1742:L P[1218]  R[157] mm/sec CNT100 Offset,PR[24:Rotate_Offset] ;
1743:L P[1219]  R[157] mm/sec CNT100 Offset,PR[24:Rotate_Offset] ;
1744:L P[1220]  R[157] mm/sec CNT100 Offset,PR[24:Rotate_Offset] ;
1745:L P[1221]  R[157] mm/sec CNT100 Offset,PR[24:Rotate_Offset] ;
1746:L P[1222]  R[157] mm/sec CNT100 Offset,PR[24:Rotate_Offset] ;
1747:L P[1223]  R[157] mm/sec CNT100 Offset,PR[24:Rotate_Offset] ;
1748: !Pass74 ;
1749: LBL[174:Pass74] ;
1750:L P[1224]  R[157] mm/sec FINE Offset,PR[78:Offst_apprch]  ;
1751: WAIT   0.20(sec) ;
1752:L P[1224]  R[157] mm/sec CNT100 TA    0.00sec,CALL RUN_LASER_START Offset,PR[25:Start_Offset] ;
1754:L P[1225]  R[157] mm/sec CNT100 Offset,PR[24:Rotate_Offset] ;
1755:L P[1226]  R[157] mm/sec CNT100 TA    0.00sec,CALL RUN_LASER_STOP Offset,PR[26:Stop_Offset] ;
1757:L P[1226]  R[157] mm/sec FINE Offset,PR[76:Offst_dprt] ;
1758:L P[1227]  R[157] mm/sec CNT100 Offset,PR[24:Rotate_Offset] ;
1759:L P[1228]  R[157] mm/sec CNT100 Offset,PR[24:Rotate_Offset] ;
1760:L P[1229]  R[157] mm/sec CNT100 Offset,PR[24:Rotate_Offset] ;
1761:L P[1230]  R[157] mm/sec CNT100 Offset,PR[24:Rotate_Offset] ;
1762:L P[1231]  R[157] mm/sec CNT100 Offset,PR[24:Rotate_Offset] ;
1763:L P[1232]  R[157] mm/sec CNT100 Offset,PR[24:Rotate_Offset] ;
1764: !Pass75 ;
1765: LBL[175:Pass75] ;
1766:L P[1233]  R[157] mm/sec FINE Offset,PR[78:Offst_apprch]  ;
1767: WAIT   0.20(sec) ;
1768:L P[1233]  R[157] mm/sec CNT100 TA    0.00sec,CALL RUN_LASER_START Offset,PR[25:Start_Offset] ;
1770:L P[1234]  R[157] mm/sec CNT100 Offset,PR[24:Rotate_Offset] ;
1771:L P[1235]  R[157] mm/sec CNT100 TA    0.00sec,CALL RUN_LASER_STOP Offset,PR[26:Stop_Offset] ;
1773:L P[1235]  R[157] mm/sec FINE Offset,PR[76:Offst_dprt] ;
1774:L P[1236]  R[157] mm/sec CNT100 Offset,PR[24:Rotate_Offset] ;
1775:L P[1237]  R[157] mm/sec CNT100 Offset,PR[24:Rotate_Offset] ;
1776:L P[1238]  R[157] mm/sec CNT100 Offset,PR[24:Rotate_Offset] ;
1777:L P[1239]  R[157] mm/sec CNT100 Offset,PR[24:Rotate_Offset] ;
1778:L P[1240]  R[157] mm/sec CNT100 Offset,PR[24:Rotate_Offset] ;
1779:L P[1241]  R[157] mm/sec CNT100 Offset,PR[24:Rotate_Offset] ;
1780: !Pass76 ;
1781: LBL[176:Pass76] ;
1782:L P[1242]  R[157] mm/sec FINE Offset,PR[78:Offst_apprch]  ;
1783: WAIT   0.20(sec) ;
1784:L P[1242]  R[157] mm/sec CNT100 TA    0.00sec,CALL RUN_LASER_START Offset,PR[25:Start_Offset] ;
1786:L P[1243]  R[157] mm/sec CNT100 Offset,PR[24:Rotate_Offset] ;
1787:L P[1244]  R[157] mm/sec CNT100 Offset,PR[24:Rotate_Offset] ;
1788:L P[1245]  R[157] mm/sec CNT100 Offset,PR[24:Rotate_Offset] ;
1789:L P[1246]  R[157] mm/sec CNT100 Offset,PR[24:Rotate_Offset] ;
1790:L P[1247]  R[157] mm/sec CNT100 TA    0.00sec,CALL RUN_LASER_STOP Offset,PR[26:Stop_Offset] ;
1792:L P[1247]  R[157] mm/sec FINE Offset,PR[76:Offst_dprt] ;
1793:L P[1248]  R[157] mm/sec CNT100 Offset,PR[24:Rotate_Offset] ;
1794:L P[1249]  R[157] mm/sec CNT100 Offset,PR[24:Rotate_Offset] ;
1795:L P[1250]  R[157] mm/sec CNT100 Offset,PR[24:Rotate_Offset] ;
1796:L P[1251]  R[157] mm/sec CNT100 Offset,PR[24:Rotate_Offset] ;
1797:L P[1252]  R[157] mm/sec CNT100 Offset,PR[24:Rotate_Offset] ;
1798:L P[1253]  R[157] mm/sec CNT100 Offset,PR[24:Rotate_Offset] ;
1799: !Pass77 ;
1800: LBL[177:Pass77] ;
1801:L P[1254]  R[157] mm/sec FINE Offset,PR[78:Offst_apprch]  ;
1802: WAIT   0.20(sec) ;
1803:L P[1254]  R[157] mm/sec CNT100 TA    0.00sec,CALL RUN_LASER_START Offset,PR[25:Start_Offset] ;
1805:L P[1255]  R[157] mm/sec CNT100 Offset,PR[24:Rotate_Offset] ;
1806:L P[1256]  R[157] mm/sec CNT100 TA    0.00sec,CALL RUN_LASER_STOP Offset,PR[26:Stop_Offset] ;
1808:L P[1256]  R[157] mm/sec FINE Offset,PR[76:Offst_dprt] ;
1809:L P[1257]  R[157] mm/sec CNT100 Offset,PR[24:Rotate_Offset] ;
1810:L P[1258]  R[157] mm/sec CNT100 Offset,PR[24:Rotate_Offset] ;
1811:L P[1259]  R[157] mm/sec CNT100 Offset,PR[24:Rotate_Offset] ;
1812:L P[1260]  R[157] mm/sec CNT100 Offset,PR[24:Rotate_Offset] ;
1813:L P[1261]  R[157] mm/sec CNT100 Offset,PR[24:Rotate_Offset] ;
1814:L P[1262]  R[157] mm/sec CNT100 Offset,PR[24:Rotate_Offset] ;
1815: !Pass78 ;
1816: LBL[178:Pass78] ;
1817:L P[1263]  R[157] mm/sec FINE Offset,PR[78:Offst_apprch]  ;
1818: WAIT   0.20(sec) ;
1819:L P[1263]  R[157] mm/sec CNT100 TA    0.00sec,CALL RUN_LASER_START Offset,PR[25:Start_Offset] ;
1821:L P[1264]  R[157] mm/sec CNT100 Offset,PR[24:Rotate_Offset] ;
1822:L P[1265]  R[157] mm/sec CNT100 TA    0.00sec,CALL RUN_LASER_STOP Offset,PR[26:Stop_Offset] ;
1824:L P[1265]  R[157] mm/sec FINE Offset,PR[76:Offst_dprt] ;
1825:L P[1266]  R[157] mm/sec CNT100 Offset,PR[24:Rotate_Offset] ;
1826:L P[1267]  R[157] mm/sec CNT100 Offset,PR[24:Rotate_Offset] ;
1827:L P[1268]  R[157] mm/sec CNT100 Offset,PR[24:Rotate_Offset] ;
1828:L P[1269]  R[157] mm/sec CNT100 Offset,PR[24:Rotate_Offset] ;
1829:L P[1270]  R[157] mm/sec CNT100 Offset,PR[24:Rotate_Offset] ;
1830:L P[1271]  R[157] mm/sec CNT100 Offset,PR[24:Rotate_Offset] ;
1831: !Pass79 ;
1832: LBL[179:Pass79] ;
1833:L P[1272]  R[157] mm/sec FINE Offset,PR[78:Offst_apprch]  ;
1834: WAIT   0.20(sec) ;
1835:L P[1272]  R[157] mm/sec CNT100 TA    0.00sec,CALL RUN_LASER_START Offset,PR[25:Start_Offset] ;
1837:L P[1273]  R[157] mm/sec CNT100 Offset,PR[24:Rotate_Offset] ;
1838:L P[1274]  R[157] mm/sec CNT100 TA    0.00sec,CALL RUN_LASER_STOP Offset,PR[26:Stop_Offset] ;
1840:L P[1274]  R[157] mm/sec FINE Offset,PR[76:Offst_dprt] ;
1841:L P[1275]  R[157] mm/sec CNT100 Offset,PR[24:Rotate_Offset] ;
1842:L P[1276]  R[157] mm/sec CNT100 Offset,PR[24:Rotate_Offset] ;
1843:L P[1277]  R[157] mm/sec CNT100 Offset,PR[24:Rotate_Offset] ;
1844:L P[1278]  R[157] mm/sec CNT100 Offset,PR[24:Rotate_Offset] ;
1845:L P[1279]  R[157] mm/sec CNT100 Offset,PR[24:Rotate_Offset] ;
1846:L P[1280]  R[157] mm/sec CNT100 Offset,PR[24:Rotate_Offset] ;
1847: !Pass80 ;
1848: LBL[180:Pass80] ;
1849:L P[1281]  R[157] mm/sec FINE Offset,PR[78:Offst_apprch]  ;
1850: WAIT   0.20(sec) ;
1851:L P[1281]  R[157] mm/sec CNT100 TA    0.00sec,CALL RUN_LASER_START Offset,PR[25:Start_Offset] ;
1853:L P[1282]  R[157] mm/sec CNT100 Offset,PR[24:Rotate_Offset] ;
1854:L P[1283]  R[157] mm/sec CNT100 TA    0.00sec,CALL RUN_LASER_STOP Offset,PR[26:Stop_Offset] ;
1856:L P[1283]  R[157] mm/sec FINE Offset,PR[76:Offst_dprt] ;
1857:L P[1284]  R[157] mm/sec CNT100 Offset,PR[24:Rotate_Offset] ;
1858:L P[1285]  R[157] mm/sec CNT100 Offset,PR[24:Rotate_Offset] ;
1859:L P[1286]  R[157] mm/sec CNT100 Offset,PR[24:Rotate_Offset] ;
1860:L P[1287]  R[157] mm/sec CNT100 Offset,PR[24:Rotate_Offset] ;
1861:L P[1288]  R[157] mm/sec CNT100 Offset,PR[24:Rotate_Offset] ;
1862:L P[1289]  R[157] mm/sec CNT100 Offset,PR[24:Rotate_Offset] ;
1863: !Pass81 ;
1864: LBL[181:Pass81] ;
1865:L P[1290]  R[157] mm/sec FINE Offset,PR[78:Offst_apprch]  ;
1866: WAIT   0.20(sec) ;
1867:L P[1290]  R[157] mm/sec CNT100 TA    0.00sec,CALL RUN_LASER_START Offset,PR[25:Start_Offset] ;
1869:L P[1291]  R[157] mm/sec CNT100 Offset,PR[24:Rotate_Offset] ;
1870:L P[1292]  R[157] mm/sec CNT100 TA    0.00sec,CALL RUN_LASER_STOP Offset,PR[26:Stop_Offset] ;
1872:L P[1292]  R[157] mm/sec FINE Offset,PR[76:Offst_dprt] ;
1873:L P[1293]  R[157] mm/sec CNT100 Offset,PR[24:Rotate_Offset] ;
1874:L P[1294]  R[157] mm/sec CNT100 Offset,PR[24:Rotate_Offset] ;
1875:L P[1295]  R[157] mm/sec CNT100 Offset,PR[24:Rotate_Offset] ;
1876:L P[1296]  R[157] mm/sec CNT100 Offset,PR[24:Rotate_Offset] ;
1877:L P[1297]  R[157] mm/sec CNT100 Offset,PR[24:Rotate_Offset] ;
1878:L P[1298]  R[157] mm/sec CNT100 Offset,PR[24:Rotate_Offset] ;
1879: !Pass82 ;
1880: LBL[182:Pass82] ;
1881:L P[1299]  R[157] mm/sec FINE Offset,PR[78:Offst_apprch]  ;
1882: WAIT   0.20(sec) ;
1883:L P[1299]  R[157] mm/sec CNT100 TA    0.00sec,CALL RUN_LASER_START Offset,PR[25:Start_Offset] ;
1885:L P[1300]  R[157] mm/sec CNT100 Offset,PR[24:Rotate_Offset] ;
1886:L P[1301]  R[157] mm/sec CNT100 TA    0.00sec,CALL RUN_LASER_STOP Offset,PR[26:Stop_Offset] ;
1888:L P[1301]  R[157] mm/sec FINE Offset,PR[76:Offst_dprt] ;
1889:L P[1302]  R[157] mm/sec CNT100 Offset,PR[24:Rotate_Offset] ;
1890:L P[1303]  R[157] mm/sec CNT100 Offset,PR[24:Rotate_Offset] ;
1891:L P[1304]  R[157] mm/sec CNT100 Offset,PR[24:Rotate_Offset] ;
1892:L P[1305]  R[157] mm/sec CNT100 Offset,PR[24:Rotate_Offset] ;
1893:L P[1306]  R[157] mm/sec CNT100 Offset,PR[24:Rotate_Offset] ;
1894:L P[1307]  R[157] mm/sec CNT100 Offset,PR[24:Rotate_Offset] ;
1895: !Pass83 ;
1896: LBL[183:Pass83] ;
1897:L P[1308]  R[157] mm/sec FINE Offset,PR[78:Offst_apprch]  ;
1898: WAIT   0.20(sec) ;
1899:L P[1308]  R[157] mm/sec CNT100 TA    0.00sec,CALL RUN_LASER_START Offset,PR[25:Start_Offset] ;
1901:L P[1309]  R[157] mm/sec CNT100 Offset,PR[24:Rotate_Offset] ;
1902:L P[1310]  R[157] mm/sec CNT100 Offset,PR[24:Rotate_Offset] ;
1903:L P[1311]  R[157] mm/sec CNT100 Offset,PR[24:Rotate_Offset] ;
1904:L P[1312]  R[157] mm/sec CNT100 TA    0.00sec,CALL RUN_LASER_STOP Offset,PR[26:Stop_Offset] ;
1906:L P[1312]  R[157] mm/sec FINE Offset,PR[76:Offst_dprt] ;
1907:L P[1313]  R[157] mm/sec CNT100 Offset,PR[24:Rotate_Offset] ;
1908:L P[1314]  R[157] mm/sec CNT100 Offset,PR[24:Rotate_Offset] ;
1909:L P[1315]  R[157] mm/sec CNT100 Offset,PR[24:Rotate_Offset] ;
1910:L P[1316]  R[157] mm/sec CNT100 Offset,PR[24:Rotate_Offset] ;
1911:L P[1317]  R[157] mm/sec CNT100 Offset,PR[24:Rotate_Offset] ;
1912:L P[1318]  R[157] mm/sec CNT100 Offset,PR[24:Rotate_Offset] ;
1913: !Pass84 ;
1914: LBL[184:Pass84] ;
1915:L P[1319]  R[157] mm/sec FINE Offset,PR[78:Offst_apprch]  ;
1916: WAIT   0.20(sec) ;
1917:L P[1319]  R[157] mm/sec CNT100 TA    0.00sec,CALL RUN_LASER_START Offset,PR[25:Start_Offset] ;
1919:L P[1320]  R[157] mm/sec CNT100 Offset,PR[24:Rotate_Offset] ;
1920:L P[1321]  R[157] mm/sec CNT100 TA    0.00sec,CALL RUN_LASER_STOP Offset,PR[26:Stop_Offset] ;
1922:L P[1321]  R[157] mm/sec FINE Offset,PR[76:Offst_dprt] ;
1923:L P[1322]  R[157] mm/sec CNT100 Offset,PR[24:Rotate_Offset] ;
1924:L P[1323]  R[157] mm/sec CNT100 Offset,PR[24:Rotate_Offset] ;
1925:L P[1324]  R[157] mm/sec CNT100 Offset,PR[24:Rotate_Offset] ;
1926:L P[1325]  R[157] mm/sec CNT100 Offset,PR[24:Rotate_Offset] ;
1927:L P[1326]  R[157] mm/sec CNT100 Offset,PR[24:Rotate_Offset] ;
1928:L P[1327]  R[157] mm/sec CNT100 Offset,PR[24:Rotate_Offset] ;
1929: !Pass85 ;
1930: LBL[185:Pass85] ;
1931:L P[1328]  R[157] mm/sec FINE Offset,PR[78:Offst_apprch]  ;
1932: WAIT   0.20(sec) ;
1933:L P[1328]  R[157] mm/sec CNT100 TA    0.00sec,CALL RUN_LASER_START Offset,PR[25:Start_Offset] ;
1935:L P[1329]  R[157] mm/sec CNT100 Offset,PR[24:Rotate_Offset] ;
1936:L P[1330]  R[157] mm/sec CNT100 TA    0.00sec,CALL RUN_LASER_STOP Offset,PR[26:Stop_Offset] ;
1938:L P[1330]  R[157] mm/sec FINE Offset,PR[76:Offst_dprt] ;
1939:L P[1331]  R[157] mm/sec CNT100 Offset,PR[24:Rotate_Offset] ;
1940:L P[1332]  R[157] mm/sec CNT100 Offset,PR[24:Rotate_Offset] ;
1941:L P[1333]  R[157] mm/sec CNT100 Offset,PR[24:Rotate_Offset] ;
1942:L P[1334]  R[157] mm/sec CNT100 Offset,PR[24:Rotate_Offset] ;
1943:L P[1335]  R[157] mm/sec CNT100 Offset,PR[24:Rotate_Offset] ;
1944:L P[1336]  R[157] mm/sec CNT100 Offset,PR[24:Rotate_Offset] ;
1945: !Pass86 ;
1946: LBL[186:Pass86] ;
1947:L P[1337]  R[157] mm/sec FINE Offset,PR[78:Offst_apprch]  ;
1948: WAIT   0.20(sec) ;
1949:L P[1337]  R[157] mm/sec CNT100 TA    0.00sec,CALL RUN_LASER_START Offset,PR[25:Start_Offset] ;
1951:L P[1338]  R[157] mm/sec CNT100 Offset,PR[24:Rotate_Offset] ;
1952:L P[1339]  R[157] mm/sec CNT100 TA    0.00sec,CALL RUN_LASER_STOP Offset,PR[26:Stop_Offset] ;
1954:L P[1339]  R[157] mm/sec FINE Offset,PR[76:Offst_dprt] ;
1955:L P[1340]  R[157] mm/sec CNT100 Offset,PR[24:Rotate_Offset] ;
1956:L P[1341]  R[157] mm/sec CNT100 Offset,PR[24:Rotate_Offset] ;
1957:L P[1342]  R[157] mm/sec CNT100 Offset,PR[24:Rotate_Offset] ;
1958:L P[1343]  R[157] mm/sec CNT100 Offset,PR[24:Rotate_Offset] ;
1959:L P[1344]  R[157] mm/sec CNT100 Offset,PR[24:Rotate_Offset] ;
1960:L P[1345]  R[157] mm/sec CNT100 Offset,PR[24:Rotate_Offset] ;
1961: !Pass87 ;
1962: LBL[187:Pass87] ;
1963:L P[1346]  R[157] mm/sec FINE Offset,PR[78:Offst_apprch]  ;
1964: WAIT   0.20(sec) ;
1965:L P[1346]  R[157] mm/sec CNT100 TA    0.00sec,CALL RUN_LASER_START Offset,PR[25:Start_Offset] ;
1967:L P[1347]  R[157] mm/sec CNT100 Offset,PR[24:Rotate_Offset] ;
1968:L P[1348]  R[157] mm/sec CNT100 TA    0.00sec,CALL RUN_LASER_STOP Offset,PR[26:Stop_Offset] ;
1970:L P[1348]  R[157] mm/sec FINE Offset,PR[76:Offst_dprt] ;
1971:L P[1349]  R[157] mm/sec CNT100 Offset,PR[24:Rotate_Offset] ;
1972:L P[1350]  R[157] mm/sec CNT100 Offset,PR[24:Rotate_Offset] ;
1973:L P[1351]  R[157] mm/sec CNT100 Offset,PR[24:Rotate_Offset] ;
1974:L P[1352]  R[157] mm/sec CNT100 Offset,PR[24:Rotate_Offset] ;
1975:L P[1353]  R[157] mm/sec CNT100 Offset,PR[24:Rotate_Offset] ;
1976:L P[1354]  R[157] mm/sec CNT100 Offset,PR[24:Rotate_Offset] ;
1977: !Pass88 ;
1978: LBL[188:Pass88] ;
1979:L P[1355]  R[157] mm/sec FINE Offset,PR[78:Offst_apprch]  ;
1980: WAIT   0.20(sec) ;
1981:L P[1355]  R[157] mm/sec CNT100 TA    0.00sec,CALL RUN_LASER_START Offset,PR[25:Start_Offset] ;
1983:L P[1356]  R[157] mm/sec CNT100 Offset,PR[24:Rotate_Offset] ;
1984:L P[1357]  R[157] mm/sec CNT100 Offset,PR[24:Rotate_Offset] ;
1985:L P[1358]  R[157] mm/sec CNT100 Offset,PR[24:Rotate_Offset] ;
1986:L P[1359]  R[157] mm/sec CNT100 Offset,PR[24:Rotate_Offset] ;
1987:L P[1360]  R[157] mm/sec CNT100 TA    0.00sec,CALL RUN_LASER_STOP Offset,PR[26:Stop_Offset] ;
1989:L P[1360]  R[157] mm/sec FINE Offset,PR[76:Offst_dprt] ;
1990:L P[1361]  R[157] mm/sec CNT100 Offset,PR[24:Rotate_Offset] ;
1991:L P[1362]  R[157] mm/sec CNT100 Offset,PR[24:Rotate_Offset] ;
1992:L P[1363]  R[157] mm/sec CNT100 Offset,PR[24:Rotate_Offset] ;
1993:L P[1364]  R[157] mm/sec CNT100 Offset,PR[24:Rotate_Offset] ;
1994:L P[1365]  R[157] mm/sec CNT100 Offset,PR[24:Rotate_Offset] ;
1995:L P[1366]  R[157] mm/sec CNT100 Offset,PR[24:Rotate_Offset] ;
1996: !Pass89 ;
1997: LBL[189:Pass89] ;
1998:L P[1367]  R[157] mm/sec FINE Offset,PR[78:Offst_apprch]  ;
1999: WAIT   0.20(sec) ;
2000:L P[1367]  R[157] mm/sec CNT100 TA    0.00sec,CALL RUN_LASER_START Offset,PR[25:Start_Offset] ;
2002:L P[1368]  R[157] mm/sec CNT100 Offset,PR[24:Rotate_Offset] ;
2003:L P[1369]  R[157] mm/sec CNT100 Offset,PR[24:Rotate_Offset] ;
2004:L P[1370]  R[157] mm/sec CNT100 Offset,PR[24:Rotate_Offset] ;
2005:L P[1371]  R[157] mm/sec CNT100 TA    0.00sec,CALL RUN_LASER_STOP Offset,PR[26:Stop_Offset] ;
2007:L P[1371]  R[157] mm/sec FINE Offset,PR[76:Offst_dprt] ;
2008:L P[1372]  R[157] mm/sec CNT100 Offset,PR[24:Rotate_Offset] ;
2009:L P[1373]  R[157] mm/sec CNT100 Offset,PR[24:Rotate_Offset] ;
2010:L P[1374]  R[157] mm/sec CNT100 Offset,PR[24:Rotate_Offset] ;
2011:L P[1375]  R[157] mm/sec CNT100 Offset,PR[24:Rotate_Offset] ;
2012:L P[1376]  R[157] mm/sec CNT100 Offset,PR[24:Rotate_Offset] ;
2013:L P[1377]  R[157] mm/sec CNT100 Offset,PR[24:Rotate_Offset] ;
2014: !Pass90 ;
2015: LBL[190:Pass90] ;
2016:L P[1378]  R[157] mm/sec FINE Offset,PR[78:Offst_apprch]  ;
2017: WAIT   0.20(sec) ;
2018:L P[1378]  R[157] mm/sec CNT100 TA    0.00sec,CALL RUN_LASER_START Offset,PR[25:Start_Offset] ;
2020:L P[1379]  R[157] mm/sec CNT100 Offset,PR[24:Rotate_Offset] ;
2021:L P[1380]  R[157] mm/sec CNT100 Offset,PR[24:Rotate_Offset] ;
2022:L P[1381]  R[157] mm/sec CNT100 Offset,PR[24:Rotate_Offset] ;
2023:L P[1382]  R[157] mm/sec CNT100 TA    0.00sec,CALL RUN_LASER_STOP Offset,PR[26:Stop_Offset] ;
2025:L P[1382]  R[157] mm/sec FINE Offset,PR[76:Offst_dprt] ;
2026:L P[1383]  R[157] mm/sec CNT100 Offset,PR[24:Rotate_Offset] ;
2027:L P[1384]  R[157] mm/sec CNT100 Offset,PR[24:Rotate_Offset] ;
2028:L P[1385]  R[157] mm/sec CNT100 Offset,PR[24:Rotate_Offset] ;
2029:L P[1386]  R[157] mm/sec CNT100 Offset,PR[24:Rotate_Offset] ;
2030:L P[1387]  R[157] mm/sec CNT100 Offset,PR[24:Rotate_Offset] ;
2031:L P[1388]  R[157] mm/sec CNT100 Offset,PR[24:Rotate_Offset] ;
2032: !Pass91 ;
2033: LBL[191:Pass91] ;
2034:L P[1389]  R[157] mm/sec FINE Offset,PR[78:Offst_apprch]  ;
2035: WAIT   0.20(sec) ;
2036:L P[1389]  R[157] mm/sec CNT100 TA    0.00sec,CALL RUN_LASER_START Offset,PR[25:Start_Offset] ;
2038:L P[1390]  R[157] mm/sec CNT100 Offset,PR[24:Rotate_Offset] ;
2039:L P[1391]  R[157] mm/sec CNT100 TA    0.00sec,CALL RUN_LASER_STOP Offset,PR[26:Stop_Offset] ;
2041:L P[1391]  R[157] mm/sec FINE Offset,PR[76:Offst_dprt] ;
2042:L P[1392]  R[157] mm/sec CNT100 Offset,PR[24:Rotate_Offset] ;
2043:L P[1393]  R[157] mm/sec CNT100 Offset,PR[24:Rotate_Offset] ;
2044:L P[1394]  R[157] mm/sec CNT100 Offset,PR[24:Rotate_Offset] ;
2045:L P[1395]  R[157] mm/sec CNT100 Offset,PR[24:Rotate_Offset] ;
2046:L P[1396]  R[157] mm/sec CNT100 Offset,PR[24:Rotate_Offset] ;
2047:L P[1397]  R[157] mm/sec CNT100 Offset,PR[24:Rotate_Offset] ;
2048: !Pass92 ;
2049: LBL[192:Pass92] ;
2050:L P[1398]  R[157] mm/sec FINE Offset,PR[78:Offst_apprch]  ;
2051: WAIT   0.20(sec) ;
2052:L P[1398]  R[157] mm/sec CNT100 TA    0.00sec,CALL RUN_LASER_START Offset,PR[25:Start_Offset] ;
2054:L P[1399]  R[157] mm/sec CNT100 Offset,PR[24:Rotate_Offset] ;
2055:L P[1400]  R[157] mm/sec CNT100 TA    0.00sec,CALL RUN_LASER_STOP Offset,PR[26:Stop_Offset] ;
2057:L P[1400]  R[157] mm/sec FINE Offset,PR[76:Offst_dprt] ;
2058:L P[1401]  R[157] mm/sec CNT100 Offset,PR[24:Rotate_Offset] ;
2059:L P[1402]  R[157] mm/sec CNT100 Offset,PR[24:Rotate_Offset] ;
2060:L P[1403]  R[157] mm/sec CNT100 Offset,PR[24:Rotate_Offset] ;
2061:L P[1404]  R[157] mm/sec CNT100 Offset,PR[24:Rotate_Offset] ;
2062:L P[1405]  R[157] mm/sec CNT100 Offset,PR[24:Rotate_Offset] ;
2063:L P[1406]  R[157] mm/sec CNT100 Offset,PR[24:Rotate_Offset] ;
2064: !Pass93 ;
2065: LBL[193:Pass93] ;
2066:L P[1407]  R[157] mm/sec FINE Offset,PR[78:Offst_apprch]  ;
2067: WAIT   0.20(sec) ;
2068:L P[1407]  R[157] mm/sec CNT100 TA    0.00sec,CALL RUN_LASER_START Offset,PR[25:Start_Offset] ;
2070:L P[1408]  R[157] mm/sec CNT100 Offset,PR[24:Rotate_Offset] ;
2071:L P[1409]  R[157] mm/sec CNT100 Offset,PR[24:Rotate_Offset] ;
2072:L P[1410]  R[157] mm/sec CNT100 Offset,PR[24:Rotate_Offset] ;
2073:L P[1411]  R[157] mm/sec CNT100 Offset,PR[24:Rotate_Offset] ;
2074:L P[1412]  R[157] mm/sec CNT100 Offset,PR[24:Rotate_Offset] ;
2075:L P[1413]  R[157] mm/sec CNT100 Offset,PR[24:Rotate_Offset] ;
2076:L P[1414]  R[157] mm/sec CNT100 Offset,PR[24:Rotate_Offset] ;
2077:L P[1415]  R[157] mm/sec CNT100 Offset,PR[24:Rotate_Offset] ;
2078:L P[1416]  R[157] mm/sec CNT100 Offset,PR[24:Rotate_Offset] ;
2079:L P[1417]  R[157] mm/sec CNT100 TA    0.00sec,CALL RUN_LASER_STOP Offset,PR[26:Stop_Offset] ;
2081:L P[1417]  R[157] mm/sec FINE Offset,PR[76:Offst_dprt] ;
2082:L P[1418]  R[157] mm/sec CNT100 Offset,PR[24:Rotate_Offset] ;
2083:L P[1419]  R[157] mm/sec CNT100 Offset,PR[24:Rotate_Offset] ;
2084:L P[1420]  R[157] mm/sec CNT100 Offset,PR[24:Rotate_Offset] ;
2085:L P[1421]  R[157] mm/sec CNT100 Offset,PR[24:Rotate_Offset] ;
2086:L P[1422]  R[157] mm/sec CNT100 Offset,PR[24:Rotate_Offset] ;
2087:L P[1423]  R[157] mm/sec CNT100 Offset,PR[24:Rotate_Offset] ;
2088: !Pass94 ;
2089: LBL[194:Pass94] ;
2090:L P[1424]  R[157] mm/sec FINE Offset,PR[78:Offst_apprch]  ;
2091: WAIT   0.20(sec) ;
2092:L P[1424]  R[157] mm/sec CNT100 TA    0.00sec,CALL RUN_LASER_START Offset,PR[25:Start_Offset] ;
2094:L P[1425]  R[157] mm/sec CNT100 Offset,PR[24:Rotate_Offset] ;
2095:L P[1426]  R[157] mm/sec CNT100 Offset,PR[24:Rotate_Offset] ;
2096:L P[1427]  R[157] mm/sec CNT100 Offset,PR[24:Rotate_Offset] ;
2097:L P[1428]  R[157] mm/sec CNT100 Offset,PR[24:Rotate_Offset] ;
2098:L P[1429]  R[157] mm/sec CNT100 TA    0.00sec,CALL RUN_LASER_STOP Offset,PR[26:Stop_Offset] ;
2100:L P[1429]  R[157] mm/sec FINE Offset,PR[76:Offst_dprt] ;
2101:L P[1430]  R[157] mm/sec CNT100 Offset,PR[24:Rotate_Offset] ;
2102:L P[1431]  R[157] mm/sec CNT100 Offset,PR[24:Rotate_Offset] ;
2103:L P[1432]  R[157] mm/sec CNT100 Offset,PR[24:Rotate_Offset] ;
2104:L P[1433]  R[157] mm/sec CNT100 Offset,PR[24:Rotate_Offset] ;
2105:L P[1434]  R[157] mm/sec CNT100 Offset,PR[24:Rotate_Offset] ;
2106:L P[1435]  R[157] mm/sec CNT100 Offset,PR[24:Rotate_Offset] ;
2107: !Pass95 ;
2108: LBL[195:Pass95] ;
2109:L P[1436]  R[157] mm/sec FINE Offset,PR[78:Offst_apprch]  ;
2110: WAIT   0.20(sec) ;
2111:L P[1436]  R[157] mm/sec CNT100 TA    0.00sec,CALL RUN_LASER_START Offset,PR[25:Start_Offset] ;
2113:L P[1437]  R[157] mm/sec CNT100 Offset,PR[24:Rotate_Offset] ;
2114:L P[1438]  R[157] mm/sec CNT100 Offset,PR[24:Rotate_Offset] ;
2115:L P[1439]  R[157] mm/sec CNT100 Offset,PR[24:Rotate_Offset] ;
2116:L P[1440]  R[157] mm/sec CNT100 TA    0.00sec,CALL RUN_LASER_STOP Offset,PR[26:Stop_Offset] ;
2118:L P[1440]  R[157] mm/sec FINE Offset,PR[76:Offst_dprt] ;
2119:L P[1441]  R[157] mm/sec CNT100 Offset,PR[24:Rotate_Offset] ;
2120:L P[1442]  R[157] mm/sec CNT100 Offset,PR[24:Rotate_Offset] ;
2121:L P[1443]  R[157] mm/sec CNT100 Offset,PR[24:Rotate_Offset] ;
2122:L P[1444]  R[157] mm/sec CNT100 Offset,PR[24:Rotate_Offset] ;
2123:L P[1445]  R[157] mm/sec CNT100 Offset,PR[24:Rotate_Offset] ;
2124:L P[1446]  R[157] mm/sec CNT100 Offset,PR[24:Rotate_Offset] ;
2125: !Pass96 ;
2126: LBL[196:Pass96] ;
2127:L P[1447]  R[157] mm/sec FINE Offset,PR[78:Offst_apprch]  ;
2128: WAIT   0.20(sec) ;
2129:L P[1447]  R[157] mm/sec CNT100 TA    0.00sec,CALL RUN_LASER_START Offset,PR[25:Start_Offset] ;
2131:L P[1448]  R[157] mm/sec CNT100 Offset,PR[24:Rotate_Offset] ;
2132:L P[1449]  R[157] mm/sec CNT100 Offset,PR[24:Rotate_Offset] ;
2133:L P[1450]  R[157] mm/sec CNT100 Offset,PR[24:Rotate_Offset] ;
2134:L P[1451]  R[157] mm/sec CNT100 TA    0.00sec,CALL RUN_LASER_STOP Offset,PR[26:Stop_Offset] ;
2136:L P[1451]  R[157] mm/sec FINE Offset,PR[76:Offst_dprt] ;
2137:L P[1452]  R[157] mm/sec CNT100 Offset,PR[24:Rotate_Offset] ;
2138:L P[1453]  R[157] mm/sec CNT100 Offset,PR[24:Rotate_Offset] ;
2139:L P[1454]  R[157] mm/sec CNT100 Offset,PR[24:Rotate_Offset] ;
2140:L P[1455]  R[157] mm/sec CNT100 Offset,PR[24:Rotate_Offset] ;
2141:L P[1456]  R[157] mm/sec CNT100 Offset,PR[24:Rotate_Offset] ;
2142:L P[1457]  R[157] mm/sec CNT100 Offset,PR[24:Rotate_Offset] ;
2143: !Pass97 ;
2144: LBL[197:Pass97] ;
2145:L P[1458]  R[157] mm/sec FINE Offset,PR[78:Offst_apprch]  ;
2146: WAIT   0.20(sec) ;
2147:L P[1458]  R[157] mm/sec CNT100 TA    0.00sec,CALL RUN_LASER_START Offset,PR[25:Start_Offset] ;
2149:L P[1459]  R[157] mm/sec CNT100 Offset,PR[24:Rotate_Offset] ;
2150:L P[1460]  R[157] mm/sec CNT100 Offset,PR[24:Rotate_Offset] ;
2151:L P[1461]  R[157] mm/sec CNT100 Offset,PR[24:Rotate_Offset] ;
2152:L P[1462]  R[157] mm/sec CNT100 TA    0.00sec,CALL RUN_LASER_STOP Offset,PR[26:Stop_Offset] ;
2154:L P[1462]  R[157] mm/sec FINE Offset,PR[76:Offst_dprt] ;
2155:L P[1463]  R[157] mm/sec CNT100 Offset,PR[24:Rotate_Offset] ;
2156:L P[1464]  R[157] mm/sec CNT100 Offset,PR[24:Rotate_Offset] ;
2157:L P[1465]  R[157] mm/sec CNT100 Offset,PR[24:Rotate_Offset] ;
2158:L P[1466]  R[157] mm/sec CNT100 Offset,PR[24:Rotate_Offset] ;
2159:L P[1467]  R[157] mm/sec CNT100 Offset,PR[24:Rotate_Offset] ;
2160:L P[1468]  R[157] mm/sec CNT100 Offset,PR[24:Rotate_Offset] ;
2161: !Pass98 ;
2162: LBL[198:Pass98] ;
2163:L P[1469]  R[157] mm/sec FINE Offset,PR[78:Offst_apprch]  ;
2164: WAIT   0.20(sec) ;
2165:L P[1469]  R[157] mm/sec CNT100 TA    0.00sec,CALL RUN_LASER_START Offset,PR[25:Start_Offset] ;
2167:L P[1470]  R[157] mm/sec CNT100 Offset,PR[24:Rotate_Offset] ;
2168:L P[1471]  R[157] mm/sec CNT100 Offset,PR[24:Rotate_Offset] ;
2169:L P[1472]  R[157] mm/sec CNT100 Offset,PR[24:Rotate_Offset] ;
2170:L P[1473]  R[157] mm/sec CNT100 TA    0.00sec,CALL RUN_LASER_STOP Offset,PR[26:Stop_Offset] ;
2172:L P[1473]  R[157] mm/sec FINE Offset,PR[76:Offst_dprt] ;
2173:L P[1474]  R[157] mm/sec CNT100 Offset,PR[24:Rotate_Offset] ;
2174:L P[1475]  R[157] mm/sec CNT100 Offset,PR[24:Rotate_Offset] ;
2175:L P[1476]  R[157] mm/sec CNT100 Offset,PR[24:Rotate_Offset] ;
2176:L P[1477]  R[157] mm/sec CNT100 Offset,PR[24:Rotate_Offset] ;
2177:L P[1478]  R[157] mm/sec CNT100 Offset,PR[24:Rotate_Offset] ;
2178:L P[1479]  R[157] mm/sec CNT100 Offset,PR[24:Rotate_Offset] ;
2179: !Pass99 ;
2180: LBL[199:Pass99] ;
2181:L P[1480]  R[157] mm/sec FINE Offset,PR[78:Offst_apprch]  ;
2182: WAIT   0.20(sec) ;
2183:L P[1480]  R[157] mm/sec CNT100 TA    0.00sec,CALL RUN_LASER_START Offset,PR[25:Start_Offset] ;
2185:L P[1481]  R[157] mm/sec CNT100 Offset,PR[24:Rotate_Offset] ;
2186:L P[1482]  R[157] mm/sec CNT100 TA    0.00sec,CALL RUN_LASER_STOP Offset,PR[26:Stop_Offset] ;
2188:L P[1482]  R[157] mm/sec FINE Offset,PR[76:Offst_dprt] ;
2189:L P[1483]  R[157] mm/sec CNT100 Offset,PR[24:Rotate_Offset] ;
2190:L P[1484]  R[157] mm/sec CNT100 Offset,PR[24:Rotate_Offset] ;
2191:L P[1485]  R[157] mm/sec CNT100 Offset,PR[24:Rotate_Offset] ;
2192:L P[1486]  R[157] mm/sec CNT100 Offset,PR[24:Rotate_Offset] ;
2193:L P[1487]  R[157] mm/sec CNT100 Offset,PR[24:Rotate_Offset] ;
2194:L P[1488]  R[157] mm/sec CNT100 Offset,PR[24:Rotate_Offset] ;
2195: !Pass100 ;
2196: LBL[1100:Pass100] ;
2197:L P[1489]  R[157] mm/sec FINE Offset,PR[78:Offst_apprch]  ;
2198: WAIT   0.20(sec) ;
2199:L P[1489]  R[157] mm/sec CNT100 TA    0.00sec,CALL RUN_LASER_START Offset,PR[25:Start_Offset] ;
2201:L P[1490]  R[157] mm/sec CNT100 Offset,PR[24:Rotate_Offset] ;
2202:L P[1491]  R[157] mm/sec CNT100 TA    0.00sec,CALL RUN_LASER_STOP Offset,PR[26:Stop_Offset] ;
2204:L P[1491]  R[157] mm/sec FINE Offset,PR[76:Offst_dprt] ;
2205:L P[1492]  R[157] mm/sec CNT100 Offset,PR[24:Rotate_Offset] ;
2206:L P[1493]  R[157] mm/sec CNT100 Offset,PR[24:Rotate_Offset] ;
2207:L P[1494]  R[157] mm/sec CNT100 Offset,PR[24:Rotate_Offset] ;
2208:L P[1495]  R[157] mm/sec CNT100 Offset,PR[24:Rotate_Offset] ;
2209:L P[1496]  R[157] mm/sec CNT100 Offset,PR[24:Rotate_Offset] ;
2210:L P[1497]  R[157] mm/sec CNT100 Offset,PR[24:Rotate_Offset] ;
2211: !Pass101 ;
2212: LBL[1101:Pass101] ;
2213:L P[1498]  R[157] mm/sec FINE Offset,PR[78:Offst_apprch]  ;
2214: WAIT   0.20(sec) ;
2215:L P[1498]  R[157] mm/sec CNT100 TA    0.00sec,CALL RUN_LASER_START Offset,PR[25:Start_Offset] ;
2217:L P[1499]  R[157] mm/sec CNT100 Offset,PR[24:Rotate_Offset] ;
2218:L P[1500]  R[157] mm/sec CNT100 Offset,PR[24:Rotate_Offset] ;
2219:L P[1501]  R[157] mm/sec CNT100 Offset,PR[24:Rotate_Offset] ;
2220:L P[1502]  R[157] mm/sec CNT100 TA    0.00sec,CALL RUN_LASER_STOP Offset,PR[26:Stop_Offset] ;
2222:L P[1502]  R[157] mm/sec FINE Offset,PR[76:Offst_dprt] ;
2223:L P[1503]  R[157] mm/sec CNT100 Offset,PR[24:Rotate_Offset] ;
2224:L P[1504]  R[157] mm/sec CNT100 Offset,PR[24:Rotate_Offset] ;
2225:L P[1505]  R[157] mm/sec CNT100 Offset,PR[24:Rotate_Offset] ;
2226:L P[1506]  R[157] mm/sec CNT100 Offset,PR[24:Rotate_Offset] ;
2227:L P[1507]  R[157] mm/sec CNT100 Offset,PR[24:Rotate_Offset] ;
2228:L P[1508]  R[157] mm/sec CNT100 Offset,PR[24:Rotate_Offset] ;
2229: !Pass102 ;
2230: LBL[1102:Pass102] ;
2231:L P[1509]  R[157] mm/sec FINE Offset,PR[78:Offst_apprch]  ;
2232: WAIT   0.20(sec) ;
2233:L P[1509]  R[157] mm/sec CNT100 TA    0.00sec,CALL RUN_LASER_START Offset,PR[25:Start_Offset] ;
2235:L P[1510]  R[157] mm/sec CNT100 Offset,PR[24:Rotate_Offset] ;
2236:L P[1511]  R[157] mm/sec CNT100 Offset,PR[24:Rotate_Offset] ;
2237:L P[1512]  R[157] mm/sec CNT100 Offset,PR[24:Rotate_Offset] ;
2238:L P[1513]  R[157] mm/sec CNT100 TA    0.00sec,CALL RUN_LASER_STOP Offset,PR[26:Stop_Offset] ;
2240:L P[1513]  R[157] mm/sec FINE Offset,PR[76:Offst_dprt] ;
2241:L P[1514]  R[157] mm/sec CNT100 Offset,PR[24:Rotate_Offset] ;
2242:L P[1515]  R[157] mm/sec CNT100 Offset,PR[24:Rotate_Offset] ;
2243:L P[1516]  R[157] mm/sec CNT100 Offset,PR[24:Rotate_Offset] ;
2244:L P[1517]  R[157] mm/sec CNT100 Offset,PR[24:Rotate_Offset] ;
2245:L P[1518]  R[157] mm/sec CNT100 Offset,PR[24:Rotate_Offset] ;
2246:L P[1519]  R[157] mm/sec CNT100 Offset,PR[24:Rotate_Offset] ;
2247: !Pass103 ;
2248: LBL[1103:Pass103] ;
2249:L P[1520]  R[157] mm/sec FINE Offset,PR[78:Offst_apprch]  ;
2250: WAIT   0.20(sec) ;
2251:L P[1520]  R[157] mm/sec CNT100 TA    0.00sec,CALL RUN_LASER_START Offset,PR[25:Start_Offset] ;
2253:L P[1521]  R[157] mm/sec CNT100 Offset,PR[24:Rotate_Offset] ;
2254:L P[1522]  R[157] mm/sec CNT100 Offset,PR[24:Rotate_Offset] ;
2255:L P[1523]  R[157] mm/sec CNT100 Offset,PR[24:Rotate_Offset] ;
2256:L P[1524]  R[157] mm/sec CNT100 TA    0.00sec,CALL RUN_LASER_STOP Offset,PR[26:Stop_Offset] ;
2258:L P[1524]  R[157] mm/sec FINE Offset,PR[76:Offst_dprt] ;
2259:L P[1525]  R[157] mm/sec CNT100 Offset,PR[24:Rotate_Offset] ;
2260:L P[1526]  R[157] mm/sec CNT100 Offset,PR[24:Rotate_Offset] ;
2261:L P[1527]  R[157] mm/sec CNT100 Offset,PR[24:Rotate_Offset] ;
2262:L P[1528]  R[157] mm/sec CNT100 Offset,PR[24:Rotate_Offset] ;
2263:L P[1529]  R[157] mm/sec CNT100 Offset,PR[24:Rotate_Offset] ;
2264:L P[1530]  R[157] mm/sec CNT100 Offset,PR[24:Rotate_Offset] ;
2265: !Pass104 ;
2266: LBL[1104:Pass104] ;
2267:L P[1531]  R[157] mm/sec FINE Offset,PR[78:Offst_apprch]  ;
2268: WAIT   0.20(sec) ;
2269:L P[1531]  R[157] mm/sec CNT100 TA    0.00sec,CALL RUN_LASER_START Offset,PR[25:Start_Offset] ;
2271:L P[1532]  R[157] mm/sec CNT100 Offset,PR[24:Rotate_Offset] ;
2272:L P[1533]  R[157] mm/sec CNT100 Offset,PR[24:Rotate_Offset] ;
2273:L P[1534]  R[157] mm/sec CNT100 Offset,PR[24:Rotate_Offset] ;
2274:L P[1535]  R[157] mm/sec CNT100 TA    0.00sec,CALL RUN_LASER_STOP Offset,PR[26:Stop_Offset] ;
2276:L P[1535]  R[157] mm/sec FINE Offset,PR[76:Offst_dprt] ;
2277:L P[1536]  R[157] mm/sec CNT100 Offset,PR[24:Rotate_Offset] ;
2278:L P[1537]  R[157] mm/sec CNT100 Offset,PR[24:Rotate_Offset] ;
2279:L P[1538]  R[157] mm/sec CNT100 Offset,PR[24:Rotate_Offset] ;
2280:L P[1539]  R[157] mm/sec CNT100 Offset,PR[24:Rotate_Offset] ;
2281:L P[1540]  R[157] mm/sec CNT100 Offset,PR[24:Rotate_Offset] ;
2282:L P[1541]  R[157] mm/sec CNT100 Offset,PR[24:Rotate_Offset] ;
2283: !Pass105 ;
2284: LBL[1105:Pass105] ;
2285:L P[1542]  R[157] mm/sec FINE Offset,PR[78:Offst_apprch]  ;
2286: WAIT   0.20(sec) ;
2287:L P[1542]  R[157] mm/sec CNT100 TA    0.00sec,CALL RUN_LASER_START Offset,PR[25:Start_Offset] ;
2289:L P[1543]  R[157] mm/sec CNT100 Offset,PR[24:Rotate_Offset] ;
2290:L P[1544]  R[157] mm/sec CNT100 Offset,PR[24:Rotate_Offset] ;
2291:L P[1545]  R[157] mm/sec CNT100 Offset,PR[24:Rotate_Offset] ;
2292:L P[1546]  R[157] mm/sec CNT100 Offset,PR[24:Rotate_Offset] ;
2293:L P[1547]  R[157] mm/sec CNT100 TA    0.00sec,CALL RUN_LASER_STOP Offset,PR[26:Stop_Offset] ;
2295:L P[1547]  R[157] mm/sec FINE Offset,PR[76:Offst_dprt] ;
2296:L P[1548]  R[157] mm/sec CNT100 Offset,PR[24:Rotate_Offset] ;
2297:L P[1549]  R[157] mm/sec CNT100 Offset,PR[24:Rotate_Offset] ;
2298:L P[1550]  R[157] mm/sec CNT100 Offset,PR[24:Rotate_Offset] ;
2299:L P[1551]  R[157] mm/sec CNT100 Offset,PR[24:Rotate_Offset] ;
2300:L P[1552]  R[157] mm/sec CNT100 Offset,PR[24:Rotate_Offset] ;
2301:L P[1553]  R[157] mm/sec CNT100 Offset,PR[24:Rotate_Offset] ;
2302: !Pass106 ;
2303: LBL[1106:Pass106] ;
2304:L P[1554]  R[157] mm/sec FINE Offset,PR[78:Offst_apprch]  ;
2305: WAIT   0.20(sec) ;
2306:L P[1554]  R[157] mm/sec CNT100 TA    0.00sec,CALL RUN_LASER_START Offset,PR[25:Start_Offset] ;
2308:L P[1555]  R[157] mm/sec CNT100 Offset,PR[24:Rotate_Offset] ;
2309:L P[1556]  R[157] mm/sec CNT100 Offset,PR[24:Rotate_Offset] ;
2310:L P[1557]  R[157] mm/sec CNT100 Offset,PR[24:Rotate_Offset] ;
2311:L P[1558]  R[157] mm/sec CNT100 Offset,PR[24:Rotate_Offset] ;
2312:L P[1559]  R[157] mm/sec CNT100 Offset,PR[24:Rotate_Offset] ;
2313:L P[1560]  R[157] mm/sec CNT100 Offset,PR[24:Rotate_Offset] ;
2314:L P[1561]  R[157] mm/sec CNT100 Offset,PR[24:Rotate_Offset] ;
2315:L P[1562]  R[157] mm/sec CNT100 Offset,PR[24:Rotate_Offset] ;
2316:L P[1563]  R[157] mm/sec CNT100 Offset,PR[24:Rotate_Offset] ;
2317:L P[1564]  R[157] mm/sec CNT100 Offset,PR[24:Rotate_Offset] ;
2318:L P[1565]  R[157] mm/sec CNT100 TA    0.00sec,CALL RUN_LASER_STOP Offset,PR[26:Stop_Offset] ;
2320:L P[1565]  R[157] mm/sec FINE Offset,PR[76:Offst_dprt] ;
2321:L P[1566]  R[157] mm/sec CNT100 Offset,PR[24:Rotate_Offset] ;
2322:L P[1567]  R[157] mm/sec CNT100 Offset,PR[24:Rotate_Offset] ;
2323:L P[1568]  R[157] mm/sec CNT100 Offset,PR[24:Rotate_Offset] ;
2324:L P[1569]  R[157] mm/sec CNT100 Offset,PR[24:Rotate_Offset] ;
2325:L P[1570]  R[157] mm/sec CNT100 Offset,PR[24:Rotate_Offset] ;
2326:L P[1571]  R[157] mm/sec CNT100 Offset,PR[24:Rotate_Offset] ;
2327: !Pass107 ;
2328: LBL[1107:Pass107] ;
2329:L P[1572]  R[157] mm/sec FINE Offset,PR[78:Offst_apprch]  ;
2330: WAIT   0.20(sec) ;
2331:L P[1572]  R[157] mm/sec CNT100 TA    0.00sec,CALL RUN_LASER_START Offset,PR[25:Start_Offset] ;
2333:L P[1573]  R[157] mm/sec CNT100 Offset,PR[24:Rotate_Offset] ;
2334:L P[1574]  R[157] mm/sec CNT100 TA    0.00sec,CALL RUN_LASER_STOP Offset,PR[26:Stop_Offset] ;
2336:L P[1574]  R[157] mm/sec FINE Offset,PR[76:Offst_dprt] ;
2337:L P[1575]  R[157] mm/sec CNT100 Offset,PR[24:Rotate_Offset] ;
2338:L P[1576]  R[157] mm/sec CNT100 Offset,PR[24:Rotate_Offset] ;
2339:L P[1577]  R[157] mm/sec CNT100 Offset,PR[24:Rotate_Offset] ;
2340:L P[1578]  R[157] mm/sec CNT100 Offset,PR[24:Rotate_Offset] ;
2341:L P[1579]  R[157] mm/sec CNT100 Offset,PR[24:Rotate_Offset] ;
2342:L P[1580]  R[157] mm/sec CNT100 Offset,PR[24:Rotate_Offset] ;
2343: !Pass108 ;
2344: LBL[1108:Pass108] ;
2345:L P[1581]  R[157] mm/sec FINE Offset,PR[78:Offst_apprch]  ;
2346: WAIT   0.20(sec) ;
2347:L P[1581]  R[157] mm/sec CNT100 TA    0.00sec,CALL RUN_LASER_START Offset,PR[25:Start_Offset] ;
2349:L P[1582]  R[157] mm/sec CNT100 Offset,PR[24:Rotate_Offset] ;
2350:L P[1583]  R[157] mm/sec CNT100 TA    0.00sec,CALL RUN_LASER_STOP Offset,PR[26:Stop_Offset] ;
2352:L P[1583]  R[157] mm/sec FINE Offset,PR[76:Offst_dprt] ;
2353:L P[1584]  R[157] mm/sec CNT100 Offset,PR[24:Rotate_Offset] ;
2354:L P[1585]  R[157] mm/sec CNT100 Offset,PR[24:Rotate_Offset] ;
2355:L P[1586]  R[157] mm/sec CNT100 Offset,PR[24:Rotate_Offset] ;
2356:L P[1587]  R[157] mm/sec CNT100 Offset,PR[24:Rotate_Offset] ;
2357:L P[1588]  R[157] mm/sec CNT100 Offset,PR[24:Rotate_Offset] ;
2358:L P[1589]  R[157] mm/sec CNT100 Offset,PR[24:Rotate_Offset] ;
2359: !Pass109 ;
2360: LBL[1109:Pass109] ;
2361:L P[1590]  R[157] mm/sec FINE Offset,PR[78:Offst_apprch]  ;
2362: WAIT   0.20(sec) ;
2363:L P[1590]  R[157] mm/sec CNT100 TA    0.00sec,CALL RUN_LASER_START Offset,PR[25:Start_Offset] ;
2365:L P[1591]  R[157] mm/sec CNT100 Offset,PR[24:Rotate_Offset] ;
2366:L P[1592]  R[157] mm/sec CNT100 Offset,PR[24:Rotate_Offset] ;
2367:L P[1593]  R[157] mm/sec CNT100 Offset,PR[24:Rotate_Offset] ;
2368:L P[1594]  R[157] mm/sec CNT100 Offset,PR[24:Rotate_Offset] ;
2369:L P[1595]  R[157] mm/sec CNT100 Offset,PR[24:Rotate_Offset] ;
2370:L P[1596]  R[157] mm/sec CNT100 Offset,PR[24:Rotate_Offset] ;
2371:L P[1597]  R[157] mm/sec CNT100 Offset,PR[24:Rotate_Offset] ;
2372:L P[1598]  R[157] mm/sec CNT100 TA    0.00sec,CALL RUN_LASER_STOP Offset,PR[26:Stop_Offset] ;
2374:L P[1598]  R[157] mm/sec FINE Offset,PR[76:Offst_dprt] ;
2375:L P[1599]  R[157] mm/sec CNT100 Offset,PR[24:Rotate_Offset] ;
2376:L P[1600]  R[157] mm/sec CNT100 Offset,PR[24:Rotate_Offset] ;
2377:L P[1601]  R[157] mm/sec CNT100 Offset,PR[24:Rotate_Offset] ;
2378:L P[1602]  R[157] mm/sec CNT100 Offset,PR[24:Rotate_Offset] ;
2379:L P[1603]  R[157] mm/sec CNT100 Offset,PR[24:Rotate_Offset] ;
2380:L P[1604]  R[157] mm/sec CNT100 Offset,PR[24:Rotate_Offset] ;
2381: !Pass110 ;
2382: LBL[1110:Pass110] ;
2383:L P[1605]  R[157] mm/sec FINE Offset,PR[78:Offst_apprch]  ;
2384: WAIT   0.20(sec) ;
2385:L P[1605]  R[157] mm/sec CNT100 TA    0.00sec,CALL RUN_LASER_START Offset,PR[25:Start_Offset] ;
2387:L P[1606]  R[157] mm/sec CNT100 Offset,PR[24:Rotate_Offset] ;
2388:L P[1607]  R[157] mm/sec CNT100 Offset,PR[24:Rotate_Offset] ;
2389:L P[1608]  R[157] mm/sec CNT100 Offset,PR[24:Rotate_Offset] ;
2390:L P[1609]  R[157] mm/sec CNT100 Offset,PR[24:Rotate_Offset] ;
2391:L P[1610]  R[157] mm/sec CNT100 TA    0.00sec,CALL RUN_LASER_STOP Offset,PR[26:Stop_Offset] ;
2393:L P[1610]  R[157] mm/sec FINE Offset,PR[76:Offst_dprt] ;
2394:L P[1611]  R[157] mm/sec CNT100 Offset,PR[24:Rotate_Offset] ;
2395:L P[1612]  R[157] mm/sec CNT100 Offset,PR[24:Rotate_Offset] ;
2396:L P[1613]  R[157] mm/sec CNT100 Offset,PR[24:Rotate_Offset] ;
2397:L P[1614]  R[157] mm/sec CNT100 Offset,PR[24:Rotate_Offset] ;
2398:L P[1615]  R[157] mm/sec CNT100 Offset,PR[24:Rotate_Offset] ;
2399:L P[1616]  R[157] mm/sec CNT100 Offset,PR[24:Rotate_Offset] ;
2400: !Pass111 ;
2401: LBL[1111:Pass111] ;
2402:L P[1617]  R[157] mm/sec FINE Offset,PR[78:Offst_apprch]  ;
2403: WAIT   0.20(sec) ;
2404:L P[1617]  R[157] mm/sec CNT100 TA    0.00sec,CALL RUN_LASER_START Offset,PR[25:Start_Offset] ;
2406:L P[1618]  R[157] mm/sec CNT100 Offset,PR[24:Rotate_Offset] ;
2407:L P[1619]  R[157] mm/sec CNT100 Offset,PR[24:Rotate_Offset] ;
2408:L P[1620]  R[157] mm/sec CNT100 Offset,PR[24:Rotate_Offset] ;
2409:L P[1621]  R[157] mm/sec CNT100 TA    0.00sec,CALL RUN_LASER_STOP Offset,PR[26:Stop_Offset] ;
2411:L P[1621]  R[157] mm/sec FINE Offset,PR[76:Offst_dprt] ;
2412:L P[1622]  R[157] mm/sec CNT100 Offset,PR[24:Rotate_Offset] ;
2413:L P[1623]  R[157] mm/sec CNT100 Offset,PR[24:Rotate_Offset] ;
2414:L P[1624]  R[157] mm/sec CNT100 Offset,PR[24:Rotate_Offset] ;
2415:L P[1625]  R[157] mm/sec CNT100 Offset,PR[24:Rotate_Offset] ;
2416:L P[1626]  R[157] mm/sec CNT100 Offset,PR[24:Rotate_Offset] ;
2417:L P[1627]  R[157] mm/sec CNT100 Offset,PR[24:Rotate_Offset] ;
2418: !Pass112 ;
2419: LBL[1112:Pass112] ;
2420:L P[1628]  R[157] mm/sec FINE Offset,PR[78:Offst_apprch]  ;
2421: WAIT   0.20(sec) ;
2422:L P[1628]  R[157] mm/sec CNT100 TA    0.00sec,CALL RUN_LASER_START Offset,PR[25:Start_Offset] ;
2424:L P[1629]  R[157] mm/sec CNT100 Offset,PR[24:Rotate_Offset] ;
2425:L P[1630]  R[157] mm/sec CNT100 Offset,PR[24:Rotate_Offset] ;
2426:L P[1631]  R[157] mm/sec CNT100 Offset,PR[24:Rotate_Offset] ;
2427:L P[1632]  R[157] mm/sec CNT100 TA    0.00sec,CALL RUN_LASER_STOP Offset,PR[26:Stop_Offset] ;
2429:L P[1632]  R[157] mm/sec FINE Offset,PR[76:Offst_dprt] ;
2430:L P[1633]  R[157] mm/sec CNT100 Offset,PR[24:Rotate_Offset] ;
2431:L P[1634]  R[157] mm/sec CNT100 Offset,PR[24:Rotate_Offset] ;
2432:L P[1635]  R[157] mm/sec CNT100 Offset,PR[24:Rotate_Offset] ;
2433:L P[1636]  R[157] mm/sec CNT100 Offset,PR[24:Rotate_Offset] ;
2434:L P[1637]  R[157] mm/sec CNT100 Offset,PR[24:Rotate_Offset] ;
2435:L P[1638]  R[157] mm/sec CNT100 Offset,PR[24:Rotate_Offset] ;
2436: !Pass113 ;
2437: LBL[1113:Pass113] ;
2438:L P[1639]  R[157] mm/sec FINE Offset,PR[78:Offst_apprch]  ;
2439: WAIT   0.20(sec) ;
2440:L P[1639]  R[157] mm/sec CNT100 TA    0.00sec,CALL RUN_LASER_START Offset,PR[25:Start_Offset] ;
2442:L P[1640]  R[157] mm/sec CNT100 Offset,PR[24:Rotate_Offset] ;
2443:L P[1641]  R[157] mm/sec CNT100 Offset,PR[24:Rotate_Offset] ;
2444:L P[1642]  R[157] mm/sec CNT100 Offset,PR[24:Rotate_Offset] ;
2445:L P[1643]  R[157] mm/sec CNT100 TA    0.00sec,CALL RUN_LASER_STOP Offset,PR[26:Stop_Offset] ;
2447:L P[1643]  R[157] mm/sec FINE Offset,PR[76:Offst_dprt] ;
2448:L P[1644]  R[157] mm/sec CNT100 Offset,PR[24:Rotate_Offset] ;
2449:L P[1645]  R[157] mm/sec CNT100 Offset,PR[24:Rotate_Offset] ;
2450:L P[1646]  R[157] mm/sec CNT100 Offset,PR[24:Rotate_Offset] ;
2451:L P[1647]  R[157] mm/sec CNT100 Offset,PR[24:Rotate_Offset] ;
2452:L P[1648]  R[157] mm/sec CNT100 Offset,PR[24:Rotate_Offset] ;
2453:L P[1649]  R[157] mm/sec CNT100 Offset,PR[24:Rotate_Offset] ;
2454: !Pass114 ;
2455: LBL[1114:Pass114] ;
2456:L P[1650]  R[157] mm/sec FINE Offset,PR[78:Offst_apprch]  ;
2457: WAIT   0.20(sec) ;
2458:L P[1650]  R[157] mm/sec CNT100 TA    0.00sec,CALL RUN_LASER_START Offset,PR[25:Start_Offset] ;
2460:L P[1651]  R[157] mm/sec CNT100 Offset,PR[24:Rotate_Offset] ;
2461:L P[1652]  R[157] mm/sec CNT100 Offset,PR[24:Rotate_Offset] ;
2462:L P[1653]  R[157] mm/sec CNT100 Offset,PR[24:Rotate_Offset] ;
2463:L P[1654]  R[157] mm/sec CNT100 TA    0.00sec,CALL RUN_LASER_STOP Offset,PR[26:Stop_Offset] ;
2465:L P[1654]  R[157] mm/sec FINE Offset,PR[76:Offst_dprt] ;
2466:L P[1655]  R[157] mm/sec CNT100 Offset,PR[24:Rotate_Offset] ;
2467:L P[1656]  R[157] mm/sec CNT100 Offset,PR[24:Rotate_Offset] ;
2468:L P[1657]  R[157] mm/sec CNT100 Offset,PR[24:Rotate_Offset] ;
2469:L P[1658]  R[157] mm/sec CNT100 Offset,PR[24:Rotate_Offset] ;
2470:L P[1659]  R[157] mm/sec CNT100 Offset,PR[24:Rotate_Offset] ;
2471:L P[1660]  R[157] mm/sec CNT100 Offset,PR[24:Rotate_Offset] ;
2472: !Pass115 ;
2473: LBL[1115:Pass115] ;
2474:L P[1661]  R[157] mm/sec FINE Offset,PR[78:Offst_apprch]  ;
2475: WAIT   0.20(sec) ;
2476:L P[1661]  R[157] mm/sec CNT100 TA    0.00sec,CALL RUN_LASER_START Offset,PR[25:Start_Offset] ;
2478:L P[1662]  R[157] mm/sec CNT100 Offset,PR[24:Rotate_Offset] ;
2479:L P[1663]  R[157] mm/sec CNT100 TA    0.00sec,CALL RUN_LASER_STOP Offset,PR[26:Stop_Offset] ;
2481:L P[1663]  R[157] mm/sec FINE Offset,PR[76:Offst_dprt] ;
2482:L P[1664]  R[157] mm/sec CNT100 Offset,PR[24:Rotate_Offset] ;
2483:L P[1665]  R[157] mm/sec CNT100 Offset,PR[24:Rotate_Offset] ;
2484:L P[1666]  R[157] mm/sec CNT100 Offset,PR[24:Rotate_Offset] ;
2485:L P[1667]  R[157] mm/sec CNT100 Offset,PR[24:Rotate_Offset] ;
2486:L P[1668]  R[157] mm/sec CNT100 Offset,PR[24:Rotate_Offset] ;
2487:L P[1669]  R[157] mm/sec CNT100 Offset,PR[24:Rotate_Offset] ;
2488: !Pass116 ;
2489: LBL[1116:Pass116] ;
2490:L P[1670]  R[157] mm/sec FINE Offset,PR[78:Offst_apprch]  ;
2491: WAIT   0.20(sec) ;
2492:L P[1670]  R[157] mm/sec CNT100 TA    0.00sec,CALL RUN_LASER_START Offset,PR[25:Start_Offset] ;
2494:L P[1671]  R[157] mm/sec CNT100 Offset,PR[24:Rotate_Offset] ;
2495:L P[1672]  R[157] mm/sec CNT100 TA    0.00sec,CALL RUN_LASER_STOP Offset,PR[26:Stop_Offset] ;
2497:L P[1672]  R[157] mm/sec FINE Offset,PR[76:Offst_dprt] ;
2498:L P[1673]  R[157] mm/sec CNT100 Offset,PR[24:Rotate_Offset] ;
2499:L P[1674]  R[157] mm/sec CNT100 Offset,PR[24:Rotate_Offset] ;
2500:L P[1675]  R[157] mm/sec CNT100 Offset,PR[24:Rotate_Offset] ;
2501:L P[1676]  R[157] mm/sec CNT100 Offset,PR[24:Rotate_Offset] ;
2502:L P[1677]  R[157] mm/sec CNT100 Offset,PR[24:Rotate_Offset] ;
2503:L P[1678]  R[157] mm/sec CNT100 Offset,PR[24:Rotate_Offset] ;
2504: !Pass117 ;
2505: LBL[1117:Pass117] ;
2506:L P[1679]  R[157] mm/sec FINE Offset,PR[78:Offst_apprch]  ;
2507: WAIT   0.20(sec) ;
2508:L P[1679]  R[157] mm/sec CNT100 TA    0.00sec,CALL RUN_LASER_START Offset,PR[25:Start_Offset] ;
2510:L P[1680]  R[157] mm/sec CNT100 Offset,PR[24:Rotate_Offset] ;
2511:L P[1681]  R[157] mm/sec CNT100 Offset,PR[24:Rotate_Offset] ;
2512:L P[1682]  R[157] mm/sec CNT100 Offset,PR[24:Rotate_Offset] ;
2513:L P[1683]  R[157] mm/sec CNT100 TA    0.00sec,CALL RUN_LASER_STOP Offset,PR[26:Stop_Offset] ;
2515:L P[1683]  R[157] mm/sec FINE Offset,PR[76:Offst_dprt] ;
2516:L P[1684]  R[157] mm/sec CNT100 Offset,PR[24:Rotate_Offset] ;
2517:L P[1685]  R[157] mm/sec CNT100 Offset,PR[24:Rotate_Offset] ;
2518:L P[1686]  R[157] mm/sec CNT100 Offset,PR[24:Rotate_Offset] ;
2519:L P[1687]  R[157] mm/sec CNT100 Offset,PR[24:Rotate_Offset] ;
2520:L P[1688]  R[157] mm/sec CNT100 Offset,PR[24:Rotate_Offset] ;
2521:L P[1689]  R[157] mm/sec CNT100 Offset,PR[24:Rotate_Offset] ;
2522: !Pass118 ;
2523: LBL[1118:Pass118] ;
2524:L P[1690]  R[157] mm/sec FINE Offset,PR[78:Offst_apprch]  ;
2525: WAIT   0.20(sec) ;
2526:L P[1690]  R[157] mm/sec CNT100 TA    0.00sec,CALL RUN_LASER_START Offset,PR[25:Start_Offset] ;
2528:L P[1691]  R[157] mm/sec CNT100 Offset,PR[24:Rotate_Offset] ;
2529:L P[1692]  R[157] mm/sec CNT100 Offset,PR[24:Rotate_Offset] ;
2530:L P[1693]  R[157] mm/sec CNT100 Offset,PR[24:Rotate_Offset] ;
2531:L P[1694]  R[157] mm/sec CNT100 TA    0.00sec,CALL RUN_LASER_STOP Offset,PR[26:Stop_Offset] ;
2533:L P[1694]  R[157] mm/sec FINE Offset,PR[76:Offst_dprt] ;
2534:L P[1695]  R[157] mm/sec CNT100 Offset,PR[24:Rotate_Offset] ;
2535:L P[1696]  R[157] mm/sec CNT100 Offset,PR[24:Rotate_Offset] ;
2536:L P[1697]  R[157] mm/sec CNT100 Offset,PR[24:Rotate_Offset] ;
2537:L P[1698]  R[157] mm/sec CNT100 Offset,PR[24:Rotate_Offset] ;
2538:L P[1699]  R[157] mm/sec CNT100 Offset,PR[24:Rotate_Offset] ;
2539:L P[1700]  R[157] mm/sec CNT100 Offset,PR[24:Rotate_Offset] ;
2540: !Pass119 ;
2541: LBL[1119:Pass119] ;
2542:L P[1701]  R[157] mm/sec FINE Offset,PR[78:Offst_apprch]  ;
2543: WAIT   0.20(sec) ;
2544:L P[1701]  R[157] mm/sec CNT100 TA    0.00sec,CALL RUN_LASER_START Offset,PR[25:Start_Offset] ;
2546:L P[1702]  R[157] mm/sec CNT100 Offset,PR[24:Rotate_Offset] ;
2547:L P[1703]  R[157] mm/sec CNT100 Offset,PR[24:Rotate_Offset] ;
2548:L P[1704]  R[157] mm/sec CNT100 Offset,PR[24:Rotate_Offset] ;
2549:L P[1705]  R[157] mm/sec CNT100 TA    0.00sec,CALL RUN_LASER_STOP Offset,PR[26:Stop_Offset] ;
2551:L P[1705]  R[157] mm/sec FINE Offset,PR[76:Offst_dprt] ;
2552:L P[1706]  R[157] mm/sec CNT100 Offset,PR[24:Rotate_Offset] ;
2553:L P[1707]  R[157] mm/sec CNT100 Offset,PR[24:Rotate_Offset] ;
2554:L P[1708]  R[157] mm/sec CNT100 Offset,PR[24:Rotate_Offset] ;
2555:L P[1709]  R[157] mm/sec CNT100 Offset,PR[24:Rotate_Offset] ;
2556:L P[1710]  R[157] mm/sec CNT100 Offset,PR[24:Rotate_Offset] ;
2557:L P[1711]  R[157] mm/sec CNT100 Offset,PR[24:Rotate_Offset] ;
2558: !Pass120 ;
2559: LBL[1120:Pass120] ;
2560:L P[1712]  R[157] mm/sec FINE Offset,PR[78:Offst_apprch]  ;
2561: WAIT   0.20(sec) ;
2562:L P[1712]  R[157] mm/sec CNT100 TA    0.00sec,CALL RUN_LASER_START Offset,PR[25:Start_Offset] ;
2564:L P[1713]  R[157] mm/sec CNT100 Offset,PR[24:Rotate_Offset] ;
2565:L P[1714]  R[157] mm/sec CNT100 Offset,PR[24:Rotate_Offset] ;
2566:L P[1715]  R[157] mm/sec CNT100 Offset,PR[24:Rotate_Offset] ;
2567:L P[1716]  R[157] mm/sec CNT100 TA    0.00sec,CALL RUN_LASER_STOP Offset,PR[26:Stop_Offset] ;
2569:L P[1716]  R[157] mm/sec FINE Offset,PR[76:Offst_dprt] ;
2570:L P[1717]  R[157] mm/sec CNT100 Offset,PR[24:Rotate_Offset] ;
2571:L P[1718]  R[157] mm/sec CNT100 Offset,PR[24:Rotate_Offset] ;
2572:L P[1719]  R[157] mm/sec CNT100 Offset,PR[24:Rotate_Offset] ;
2573:L P[1720]  R[157] mm/sec CNT100 Offset,PR[24:Rotate_Offset] ;
2574:L P[1721]  R[157] mm/sec CNT100 Offset,PR[24:Rotate_Offset] ;
2575:L P[1722]  R[157] mm/sec CNT100 Offset,PR[24:Rotate_Offset] ;
2576: !Pass121 ;
2577: LBL[1121:Pass121] ;
2578:L P[1723]  R[157] mm/sec FINE Offset,PR[78:Offst_apprch]  ;
2579: WAIT   0.20(sec) ;
2580:L P[1723]  R[157] mm/sec CNT100 TA    0.00sec,CALL RUN_LASER_START Offset,PR[25:Start_Offset] ;
2582:L P[1724]  R[157] mm/sec CNT100 Offset,PR[24:Rotate_Offset] ;
2583:L P[1725]  R[157] mm/sec CNT100 Offset,PR[24:Rotate_Offset] ;
2584:L P[1726]  R[157] mm/sec CNT100 Offset,PR[24:Rotate_Offset] ;
2585:L P[1727]  R[157] mm/sec CNT100 Offset,PR[24:Rotate_Offset] ;
2586:L P[1728]  R[157] mm/sec CNT100 TA    0.00sec,CALL RUN_LASER_STOP Offset,PR[26:Stop_Offset] ;
2588:L P[1728]  R[157] mm/sec FINE Offset,PR[76:Offst_dprt] ;
2589:L P[1729]  R[157] mm/sec CNT100 Offset,PR[24:Rotate_Offset] ;
2590:L P[1730]  R[157] mm/sec CNT100 Offset,PR[24:Rotate_Offset] ;
2591:L P[1731]  R[157] mm/sec CNT100 Offset,PR[24:Rotate_Offset] ;
2592:L P[1732]  R[157] mm/sec CNT100 Offset,PR[24:Rotate_Offset] ;
2593:L P[1733]  R[157] mm/sec CNT100 Offset,PR[24:Rotate_Offset] ;
2594:L P[1734]  R[157] mm/sec CNT100 Offset,PR[24:Rotate_Offset] ;
2595: !Pass122 ;
2596: LBL[1122:Pass122] ;
2597:L P[1735]  R[157] mm/sec FINE Offset,PR[78:Offst_apprch]  ;
2598: WAIT   0.20(sec) ;
2599:L P[1735]  R[157] mm/sec CNT100 TA    0.00sec,CALL RUN_LASER_START Offset,PR[25:Start_Offset] ;
2601:L P[1736]  R[157] mm/sec CNT100 Offset,PR[24:Rotate_Offset] ;
2602:L P[1737]  R[157] mm/sec CNT100 Offset,PR[24:Rotate_Offset] ;
2603:L P[1738]  R[157] mm/sec CNT100 Offset,PR[24:Rotate_Offset] ;
2604:L P[1739]  R[157] mm/sec CNT100 Offset,PR[24:Rotate_Offset] ;
2605:L P[1740]  R[157] mm/sec CNT100 Offset,PR[24:Rotate_Offset] ;
2606:L P[1741]  R[157] mm/sec CNT100 Offset,PR[24:Rotate_Offset] ;
2607:L P[1742]  R[157] mm/sec CNT100 TA    0.00sec,CALL RUN_LASER_STOP Offset,PR[26:Stop_Offset] ;
2609:L P[1742]  R[157] mm/sec FINE Offset,PR[76:Offst_dprt] ;
2610:L P[1743]  R[157] mm/sec CNT100 Offset,PR[24:Rotate_Offset] ;
2611:L P[1744]  R[157] mm/sec CNT100 Offset,PR[24:Rotate_Offset] ;
2612:L P[1745]  R[157] mm/sec CNT100 Offset,PR[24:Rotate_Offset] ;
2613:L P[1746]  R[157] mm/sec CNT100 Offset,PR[24:Rotate_Offset] ;
2614:L P[1747]  R[157] mm/sec CNT100 Offset,PR[24:Rotate_Offset] ;
2615:L P[1748]  R[157] mm/sec CNT100 Offset,PR[24:Rotate_Offset] ;
2616: !Pass123 ;
2617: LBL[1123:Pass123] ;
2618:L P[1749]  R[157] mm/sec FINE Offset,PR[78:Offst_apprch]  ;
2619: WAIT   0.20(sec) ;
2620:L P[1749]  R[157] mm/sec CNT100 TA    0.00sec,CALL RUN_LASER_START Offset,PR[25:Start_Offset] ;
2622:L P[1750]  R[157] mm/sec CNT100 Offset,PR[24:Rotate_Offset] ;
2623:L P[1751]  R[157] mm/sec CNT100 TA    0.00sec,CALL RUN_LASER_STOP Offset,PR[26:Stop_Offset] ;
2625:L P[1751]  R[157] mm/sec FINE Offset,PR[76:Offst_dprt] ;
2626:L P[1752]  R[157] mm/sec CNT100 Offset,PR[24:Rotate_Offset] ;
2627:L P[1753]  R[157] mm/sec CNT100 Offset,PR[24:Rotate_Offset] ;
2628:L P[1754]  R[157] mm/sec CNT100 Offset,PR[24:Rotate_Offset] ;
2629:L P[1755]  R[157] mm/sec CNT100 Offset,PR[24:Rotate_Offset] ;
2630:L P[1756]  R[157] mm/sec CNT100 Offset,PR[24:Rotate_Offset] ;
2631:L P[1757]  R[157] mm/sec CNT100 Offset,PR[24:Rotate_Offset] ;
2632: !Pass124 ;
2633: LBL[1124:Pass124] ;
2634:L P[1758]  R[157] mm/sec FINE Offset,PR[78:Offst_apprch]  ;
2635: WAIT   0.20(sec) ;
2636:L P[1758]  R[157] mm/sec CNT100 TA    0.00sec,CALL RUN_LASER_START Offset,PR[25:Start_Offset] ;
2638:L P[1759]  R[157] mm/sec CNT100 Offset,PR[24:Rotate_Offset] ;
2639:L P[1760]  R[157] mm/sec CNT100 TA    0.00sec,CALL RUN_LASER_STOP Offset,PR[26:Stop_Offset] ;
2641:L P[1760]  R[157] mm/sec FINE Offset,PR[76:Offst_dprt] ;
2642:L P[1761]  R[157] mm/sec CNT100 Offset,PR[24:Rotate_Offset] ;
2643:L P[1762]  R[157] mm/sec CNT100 Offset,PR[24:Rotate_Offset] ;
2644:L P[1763]  R[157] mm/sec CNT100 Offset,PR[24:Rotate_Offset] ;
2645:L P[1764]  R[157] mm/sec CNT100 Offset,PR[24:Rotate_Offset] ;
2646:L P[1765]  R[157] mm/sec CNT100 Offset,PR[24:Rotate_Offset] ;
2647:L P[1766]  R[157] mm/sec CNT100 Offset,PR[24:Rotate_Offset] ;
2648: !Pass125 ;
2649: LBL[1125:Pass125] ;
2650:L P[1767]  R[157] mm/sec FINE Offset,PR[78:Offst_apprch]  ;
2651: WAIT   0.20(sec) ;
2652:L P[1767]  R[157] mm/sec CNT100 TA    0.00sec,CALL RUN_LASER_START Offset,PR[25:Start_Offset] ;
2654:L P[1768]  R[157] mm/sec CNT100 Offset,PR[24:Rotate_Offset] ;
2655:L P[1769]  R[157] mm/sec CNT100 Offset,PR[24:Rotate_Offset] ;
2656:L P[1770]  R[157] mm/sec CNT100 Offset,PR[24:Rotate_Offset] ;
2657:L P[1771]  R[157] mm/sec CNT100 Offset,PR[24:Rotate_Offset] ;
2658:L P[1772]  R[157] mm/sec CNT100 Offset,PR[24:Rotate_Offset] ;
2659:L P[1773]  R[157] mm/sec CNT100 TA    0.00sec,CALL RUN_LASER_STOP Offset,PR[26:Stop_Offset] ;
2661:L P[1773]  R[157] mm/sec FINE Offset,PR[76:Offst_dprt] ;
2662:L P[1774]  R[157] mm/sec CNT100 Offset,PR[24:Rotate_Offset] ;
2663:L P[1775]  R[157] mm/sec CNT100 Offset,PR[24:Rotate_Offset] ;
2664:L P[1776]  R[157] mm/sec CNT100 Offset,PR[24:Rotate_Offset] ;
2665:L P[1777]  R[157] mm/sec CNT100 Offset,PR[24:Rotate_Offset] ;
2666:L P[1778]  R[157] mm/sec CNT100 Offset,PR[24:Rotate_Offset] ;
2667:L P[1779]  R[157] mm/sec CNT100 Offset,PR[24:Rotate_Offset] ;
2668: !Pass126 ;
2669: LBL[1126:Pass126] ;
2670:L P[1780]  R[157] mm/sec FINE Offset,PR[78:Offst_apprch]  ;
2671: WAIT   0.20(sec) ;
2672:L P[1780]  R[157] mm/sec CNT100 TA    0.00sec,CALL RUN_LASER_START Offset,PR[25:Start_Offset] ;
2674:L P[1781]  R[157] mm/sec CNT100 Offset,PR[24:Rotate_Offset] ;
2675:L P[1782]  R[157] mm/sec CNT100 Offset,PR[24:Rotate_Offset] ;
2676:L P[1783]  R[157] mm/sec CNT100 Offset,PR[24:Rotate_Offset] ;
2677:L P[1784]  R[157] mm/sec CNT100 Offset,PR[24:Rotate_Offset] ;
2678:L P[1785]  R[157] mm/sec CNT100 TA    0.00sec,CALL RUN_LASER_STOP Offset,PR[26:Stop_Offset] ;
2680:L P[1785]  R[157] mm/sec FINE Offset,PR[76:Offst_dprt] ;
2681:L P[1786]  R[157] mm/sec CNT100 Offset,PR[24:Rotate_Offset] ;
2682:L P[1787]  R[157] mm/sec CNT100 Offset,PR[24:Rotate_Offset] ;
2683:L P[1788]  R[157] mm/sec CNT100 Offset,PR[24:Rotate_Offset] ;
2684:L P[1789]  R[157] mm/sec CNT100 Offset,PR[24:Rotate_Offset] ;
2685:L P[1790]  R[157] mm/sec CNT100 Offset,PR[24:Rotate_Offset] ;
2686:L P[1791]  R[157] mm/sec CNT100 Offset,PR[24:Rotate_Offset] ;
2687: !Pass127 ;
2688: LBL[1127:Pass127] ;
2689:L P[1792]  R[157] mm/sec FINE Offset,PR[78:Offst_apprch]  ;
2690: WAIT   0.20(sec) ;
2691:L P[1792]  R[157] mm/sec CNT100 TA    0.00sec,CALL RUN_LASER_START Offset,PR[25:Start_Offset] ;
2693:L P[1793]  R[157] mm/sec CNT100 Offset,PR[24:Rotate_Offset] ;
2694:L P[1794]  R[157] mm/sec CNT100 Offset,PR[24:Rotate_Offset] ;
2695:L P[1795]  R[157] mm/sec CNT100 Offset,PR[24:Rotate_Offset] ;
2696:L P[1796]  R[157] mm/sec CNT100 TA    0.00sec,CALL RUN_LASER_STOP Offset,PR[26:Stop_Offset] ;
2698:L P[1796]  R[157] mm/sec FINE Offset,PR[76:Offst_dprt] ;
2699:L P[1797]  R[157] mm/sec CNT100 Offset,PR[24:Rotate_Offset] ;
2700:L P[1798]  R[157] mm/sec CNT100 Offset,PR[24:Rotate_Offset] ;
2701:L P[1799]  R[157] mm/sec CNT100 Offset,PR[24:Rotate_Offset] ;
2702:L P[1800]  R[157] mm/sec CNT100 Offset,PR[24:Rotate_Offset] ;
2703:L P[1801]  R[157] mm/sec CNT100 Offset,PR[24:Rotate_Offset] ;
2704:L P[1802]  R[157] mm/sec CNT100 Offset,PR[24:Rotate_Offset] ;
2705: !Pass128 ;
2706: LBL[1128:Pass128] ;
2707:L P[1803]  R[157] mm/sec FINE Offset,PR[78:Offst_apprch]  ;
2708: WAIT   0.20(sec) ;
2709:L P[1803]  R[157] mm/sec CNT100 TA    0.00sec,CALL RUN_LASER_START Offset,PR[25:Start_Offset] ;
2711:L P[1804]  R[157] mm/sec CNT100 Offset,PR[24:Rotate_Offset] ;
2712:L P[1805]  R[157] mm/sec CNT100 Offset,PR[24:Rotate_Offset] ;
2713:L P[1806]  R[157] mm/sec CNT100 Offset,PR[24:Rotate_Offset] ;
2714:L P[1807]  R[157] mm/sec CNT100 TA    0.00sec,CALL RUN_LASER_STOP Offset,PR[26:Stop_Offset] ;
2716:L P[1807]  R[157] mm/sec FINE Offset,PR[76:Offst_dprt] ;
2717:L P[1808]  R[157] mm/sec CNT100 Offset,PR[24:Rotate_Offset] ;
2718:L P[1809]  R[157] mm/sec CNT100 Offset,PR[24:Rotate_Offset] ;
2719:L P[1810]  R[157] mm/sec CNT100 Offset,PR[24:Rotate_Offset] ;
2720:L P[1811]  R[157] mm/sec CNT100 Offset,PR[24:Rotate_Offset] ;
2721:L P[1812]  R[157] mm/sec CNT100 Offset,PR[24:Rotate_Offset] ;
2722:L P[1813]  R[157] mm/sec CNT100 Offset,PR[24:Rotate_Offset] ;
2723: !Pass129 ;
2724: LBL[1129:Pass129] ;
2725:L P[1814]  R[157] mm/sec FINE Offset,PR[78:Offst_apprch]  ;
2726: WAIT   0.20(sec) ;
2727:L P[1814]  R[157] mm/sec CNT100 TA    0.00sec,CALL RUN_LASER_START Offset,PR[25:Start_Offset] ;
2729:L P[1815]  R[157] mm/sec CNT100 Offset,PR[24:Rotate_Offset] ;
2730:L P[1816]  R[157] mm/sec CNT100 Offset,PR[24:Rotate_Offset] ;
2731:L P[1817]  R[157] mm/sec CNT100 Offset,PR[24:Rotate_Offset] ;
2732:L P[1818]  R[157] mm/sec CNT100 TA    0.00sec,CALL RUN_LASER_STOP Offset,PR[26:Stop_Offset] ;
2734:L P[1818]  R[157] mm/sec FINE Offset,PR[76:Offst_dprt] ;
2735:L P[1819]  R[157] mm/sec CNT100 Offset,PR[24:Rotate_Offset] ;
2736:L P[1820]  R[157] mm/sec CNT100 Offset,PR[24:Rotate_Offset] ;
2737:L P[1821]  R[157] mm/sec CNT100 Offset,PR[24:Rotate_Offset] ;
2738:L P[1822]  R[157] mm/sec CNT100 Offset,PR[24:Rotate_Offset] ;
2739:L P[1823]  R[157] mm/sec CNT100 Offset,PR[24:Rotate_Offset] ;
2740:L P[1824]  R[157] mm/sec CNT100 Offset,PR[24:Rotate_Offset] ;
2741: !Pass130 ;
2742: LBL[1130:Pass130] ;
2743:L P[1825]  R[157] mm/sec FINE Offset,PR[78:Offst_apprch]  ;
2744: WAIT   0.20(sec) ;
2745:L P[1825]  R[157] mm/sec CNT100 TA    0.00sec,CALL RUN_LASER_START Offset,PR[25:Start_Offset] ;
2747:L P[1826]  R[157] mm/sec CNT100 Offset,PR[24:Rotate_Offset] ;
2748:L P[1827]  R[157] mm/sec CNT100 Offset,PR[24:Rotate_Offset] ;
2749:L P[1828]  R[157] mm/sec CNT100 Offset,PR[24:Rotate_Offset] ;
2750:L P[1829]  R[157] mm/sec CNT100 TA    0.00sec,CALL RUN_LASER_STOP Offset,PR[26:Stop_Offset] ;
2752:L P[1829]  R[157] mm/sec FINE Offset,PR[76:Offst_dprt] ;
2753:L P[1830]  R[157] mm/sec CNT100 Offset,PR[24:Rotate_Offset] ;
2754:L P[1831]  R[157] mm/sec CNT100 Offset,PR[24:Rotate_Offset] ;
2755:L P[1832]  R[157] mm/sec CNT100 Offset,PR[24:Rotate_Offset] ;
2756:L P[1833]  R[157] mm/sec CNT100 Offset,PR[24:Rotate_Offset] ;
2757:L P[1834]  R[157] mm/sec CNT100 Offset,PR[24:Rotate_Offset] ;
2758:L P[1835]  R[157] mm/sec CNT100 Offset,PR[24:Rotate_Offset] ;
2759: !Pass131 ;
2760: LBL[1131:Pass131] ;
2761:L P[1836]  R[157] mm/sec FINE Offset,PR[78:Offst_apprch]  ;
2762: WAIT   0.20(sec) ;
2763:L P[1836]  R[157] mm/sec CNT100 TA    0.00sec,CALL RUN_LASER_START Offset,PR[25:Start_Offset] ;
2765:L P[1837]  R[157] mm/sec CNT100 Offset,PR[24:Rotate_Offset] ;
2766:L P[1838]  R[157] mm/sec CNT100 TA    0.00sec,CALL RUN_LASER_STOP Offset,PR[26:Stop_Offset] ;
2768:L P[1838]  R[157] mm/sec FINE Offset,PR[76:Offst_dprt] ;
2769:L P[1839]  R[157] mm/sec CNT100 Offset,PR[24:Rotate_Offset] ;
2770:L P[1840]  R[157] mm/sec CNT100 Offset,PR[24:Rotate_Offset] ;
2771:L P[1841]  R[157] mm/sec CNT100 Offset,PR[24:Rotate_Offset] ;
2772:L P[1842]  R[157] mm/sec CNT100 Offset,PR[24:Rotate_Offset] ;
2773:L P[1843]  R[157] mm/sec CNT100 Offset,PR[24:Rotate_Offset] ;
2774:L P[1844]  R[157] mm/sec CNT100 Offset,PR[24:Rotate_Offset] ;
2775: !Pass132 ;
2776: LBL[1132:Pass132] ;
2777:L P[1845]  R[157] mm/sec FINE Offset,PR[78:Offst_apprch]  ;
2778: WAIT   0.20(sec) ;
2779:L P[1845]  R[157] mm/sec CNT100 TA    0.00sec,CALL RUN_LASER_START Offset,PR[25:Start_Offset] ;
2781:L P[1846]  R[157] mm/sec CNT100 Offset,PR[24:Rotate_Offset] ;
2782:L P[1847]  R[157] mm/sec CNT100 TA    0.00sec,CALL RUN_LASER_STOP Offset,PR[26:Stop_Offset] ;
2784:L P[1847]  R[157] mm/sec FINE Offset,PR[76:Offst_dprt] ;
2785:L P[1848]  R[157] mm/sec CNT100 Offset,PR[24:Rotate_Offset] ;
2786:L P[1849]  R[157] mm/sec CNT100 Offset,PR[24:Rotate_Offset] ;
2787:L P[1850]  R[157] mm/sec CNT100 Offset,PR[24:Rotate_Offset] ;
2788:L P[1851]  R[157] mm/sec CNT100 Offset,PR[24:Rotate_Offset] ;
2789:L P[1852]  R[157] mm/sec CNT100 Offset,PR[24:Rotate_Offset] ;
2790:L P[1853]  R[157] mm/sec CNT100 Offset,PR[24:Rotate_Offset] ;
2791: !Pass133 ;
2792: LBL[1133:Pass133] ;
2793:L P[1854]  R[157] mm/sec FINE Offset,PR[78:Offst_apprch]  ;
2794: WAIT   0.20(sec) ;
2795:L P[1854]  R[157] mm/sec CNT100 TA    0.00sec,CALL RUN_LASER_START Offset,PR[25:Start_Offset] ;
2797:L P[1855]  R[157] mm/sec CNT100 Offset,PR[24:Rotate_Offset] ;
2798:L P[1856]  R[157] mm/sec CNT100 Offset,PR[24:Rotate_Offset] ;
2799:L P[1857]  R[157] mm/sec CNT100 Offset,PR[24:Rotate_Offset] ;
2800:L P[1858]  R[157] mm/sec CNT100 TA    0.00sec,CALL RUN_LASER_STOP Offset,PR[26:Stop_Offset] ;
2802:L P[1858]  R[157] mm/sec FINE Offset,PR[76:Offst_dprt] ;
2803:L P[1859]  R[157] mm/sec CNT100 Offset,PR[24:Rotate_Offset] ;
2804:L P[1860]  R[157] mm/sec CNT100 Offset,PR[24:Rotate_Offset] ;
2805:L P[1861]  R[157] mm/sec CNT100 Offset,PR[24:Rotate_Offset] ;
2806:L P[1862]  R[157] mm/sec CNT100 Offset,PR[24:Rotate_Offset] ;
2807:L P[1863]  R[157] mm/sec CNT100 Offset,PR[24:Rotate_Offset] ;
2808:L P[1864]  R[157] mm/sec CNT100 Offset,PR[24:Rotate_Offset] ;
2809: !Pass134 ;
2810: LBL[1134:Pass134] ;
2811:L P[1865]  R[157] mm/sec FINE Offset,PR[78:Offst_apprch]  ;
2812: WAIT   0.20(sec) ;
2813:L P[1865]  R[157] mm/sec CNT100 TA    0.00sec,CALL RUN_LASER_START Offset,PR[25:Start_Offset] ;
2815:L P[1866]  R[157] mm/sec CNT100 Offset,PR[24:Rotate_Offset] ;
2816:L P[1867]  R[157] mm/sec CNT100 Offset,PR[24:Rotate_Offset] ;
2817:L P[1868]  R[157] mm/sec CNT100 Offset,PR[24:Rotate_Offset] ;
2818:L P[1869]  R[157] mm/sec CNT100 TA    0.00sec,CALL RUN_LASER_STOP Offset,PR[26:Stop_Offset] ;
2820:L P[1869]  R[157] mm/sec FINE Offset,PR[76:Offst_dprt] ;
2821:L P[1870]  R[157] mm/sec CNT100 Offset,PR[24:Rotate_Offset] ;
2822:L P[1871]  R[157] mm/sec CNT100 Offset,PR[24:Rotate_Offset] ;
2823:L P[1872]  R[157] mm/sec CNT100 Offset,PR[24:Rotate_Offset] ;
2824:L P[1873]  R[157] mm/sec CNT100 Offset,PR[24:Rotate_Offset] ;
2825:L P[1874]  R[157] mm/sec CNT100 Offset,PR[24:Rotate_Offset] ;
2826:L P[1875]  R[157] mm/sec CNT100 Offset,PR[24:Rotate_Offset] ;
2827: !Pass135 ;
2828: LBL[1135:Pass135] ;
2829:L P[1876]  R[157] mm/sec FINE Offset,PR[78:Offst_apprch]  ;
2830: WAIT   0.20(sec) ;
2831:L P[1876]  R[157] mm/sec CNT100 TA    0.00sec,CALL RUN_LASER_START Offset,PR[25:Start_Offset] ;
2833:L P[1877]  R[157] mm/sec CNT100 Offset,PR[24:Rotate_Offset] ;
2834:L P[1878]  R[157] mm/sec CNT100 Offset,PR[24:Rotate_Offset] ;
2835:L P[1879]  R[157] mm/sec CNT100 Offset,PR[24:Rotate_Offset] ;
2836:L P[1880]  R[157] mm/sec CNT100 TA    0.00sec,CALL RUN_LASER_STOP Offset,PR[26:Stop_Offset] ;
2838:L P[1880]  R[157] mm/sec FINE Offset,PR[76:Offst_dprt] ;
2839:L P[1881]  R[157] mm/sec CNT100 Offset,PR[24:Rotate_Offset] ;
2840:L P[1882]  R[157] mm/sec CNT100 Offset,PR[24:Rotate_Offset] ;
2841:L P[1883]  R[157] mm/sec CNT100 Offset,PR[24:Rotate_Offset] ;
2842:L P[1884]  R[157] mm/sec CNT100 Offset,PR[24:Rotate_Offset] ;
2843:L P[1885]  R[157] mm/sec CNT100 Offset,PR[24:Rotate_Offset] ;
2844:L P[1886]  R[157] mm/sec CNT100 Offset,PR[24:Rotate_Offset] ;
2845: !Pass136 ;
2846: LBL[1136:Pass136] ;
2847:L P[1887]  R[157] mm/sec FINE Offset,PR[78:Offst_apprch]  ;
2848: WAIT   0.20(sec) ;
2849:L P[1887]  R[157] mm/sec CNT100 TA    0.00sec,CALL RUN_LASER_START Offset,PR[25:Start_Offset] ;
2851:L P[1888]  R[157] mm/sec CNT100 Offset,PR[24:Rotate_Offset] ;
2852:L P[1889]  R[157] mm/sec CNT100 Offset,PR[24:Rotate_Offset] ;
2853:L P[1890]  R[157] mm/sec CNT100 Offset,PR[24:Rotate_Offset] ;
2854:L P[1891]  R[157] mm/sec CNT100 TA    0.00sec,CALL RUN_LASER_STOP Offset,PR[26:Stop_Offset] ;
2856:L P[1891]  R[157] mm/sec FINE Offset,PR[76:Offst_dprt] ;
2857:L P[1892]  R[157] mm/sec CNT100 Offset,PR[24:Rotate_Offset] ;
2858:L P[1893]  R[157] mm/sec CNT100 Offset,PR[24:Rotate_Offset] ;
2859:L P[1894]  R[157] mm/sec CNT100 Offset,PR[24:Rotate_Offset] ;
2860:L P[1895]  R[157] mm/sec CNT100 Offset,PR[24:Rotate_Offset] ;
2861:L P[1896]  R[157] mm/sec CNT100 Offset,PR[24:Rotate_Offset] ;
2862:L P[1897]  R[157] mm/sec CNT100 Offset,PR[24:Rotate_Offset] ;
2863: !Pass137 ;
2864: LBL[1137:Pass137] ;
2865:L P[1898]  R[157] mm/sec FINE Offset,PR[78:Offst_apprch]  ;
2866: WAIT   0.20(sec) ;
2867:L P[1898]  R[157] mm/sec CNT100 TA    0.00sec,CALL RUN_LASER_START Offset,PR[25:Start_Offset] ;
2869:L P[1899]  R[157] mm/sec CNT100 Offset,PR[24:Rotate_Offset] ;
2870:L P[1900]  R[157] mm/sec CNT100 Offset,PR[24:Rotate_Offset] ;
2871:L P[1901]  R[157] mm/sec CNT100 Offset,PR[24:Rotate_Offset] ;
2872:L P[1902]  R[157] mm/sec CNT100 Offset,PR[24:Rotate_Offset] ;
2873:L P[1903]  R[157] mm/sec CNT100 TA    0.00sec,CALL RUN_LASER_STOP Offset,PR[26:Stop_Offset] ;
2875:L P[1903]  R[157] mm/sec FINE Offset,PR[76:Offst_dprt] ;
2876:L P[1904]  R[157] mm/sec CNT100 Offset,PR[24:Rotate_Offset] ;
2877:L P[1905]  R[157] mm/sec CNT100 Offset,PR[24:Rotate_Offset] ;
2878:L P[1906]  R[157] mm/sec CNT100 Offset,PR[24:Rotate_Offset] ;
2879:L P[1907]  R[157] mm/sec CNT100 Offset,PR[24:Rotate_Offset] ;
2880:L P[1908]  R[157] mm/sec CNT100 Offset,PR[24:Rotate_Offset] ;
2881:L P[1909]  R[157] mm/sec CNT100 Offset,PR[24:Rotate_Offset] ;
2882: !Pass138 ;
2883: LBL[1138:Pass138] ;
2884:L P[1910]  R[157] mm/sec FINE Offset,PR[78:Offst_apprch]  ;
2885: WAIT   0.20(sec) ;
2886:L P[1910]  R[157] mm/sec CNT100 TA    0.00sec,CALL RUN_LASER_START Offset,PR[25:Start_Offset] ;
2888:L P[1911]  R[157] mm/sec CNT100 Offset,PR[24:Rotate_Offset] ;
2889:L P[1912]  R[157] mm/sec CNT100 Offset,PR[24:Rotate_Offset] ;
2890:L P[1913]  R[157] mm/sec CNT100 Offset,PR[24:Rotate_Offset] ;
2891:L P[1914]  R[157] mm/sec CNT100 Offset,PR[24:Rotate_Offset] ;
2892:L P[1915]  R[157] mm/sec CNT100 Offset,PR[24:Rotate_Offset] ;
2893:L P[1916]  R[157] mm/sec CNT100 TA    0.00sec,CALL RUN_LASER_STOP Offset,PR[26:Stop_Offset] ;
2895:L P[1916]  R[157] mm/sec FINE Offset,PR[76:Offst_dprt] ;
2896:L P[1917]  R[157] mm/sec CNT100 Offset,PR[24:Rotate_Offset] ;
2897:L P[1918]  R[157] mm/sec CNT100 Offset,PR[24:Rotate_Offset] ;
2898:L P[1919]  R[157] mm/sec CNT100 Offset,PR[24:Rotate_Offset] ;
2899:L P[1920]  R[157] mm/sec CNT100 Offset,PR[24:Rotate_Offset] ;
2900:L P[1921]  R[157] mm/sec CNT100 Offset,PR[24:Rotate_Offset] ;
2901:L P[1922]  R[157] mm/sec CNT100 Offset,PR[24:Rotate_Offset] ;
2902: !Pass139 ;
2903: LBL[1139:Pass139] ;
2904:L P[1923]  R[157] mm/sec FINE Offset,PR[78:Offst_apprch]  ;
2905: WAIT   0.20(sec) ;
2906:L P[1923]  R[157] mm/sec CNT100 TA    0.00sec,CALL RUN_LASER_START Offset,PR[25:Start_Offset] ;
2908:L P[1924]  R[157] mm/sec CNT100 Offset,PR[24:Rotate_Offset] ;
2909:L P[1925]  R[157] mm/sec CNT100 TA    0.00sec,CALL RUN_LASER_STOP Offset,PR[26:Stop_Offset] ;
2911:L P[1925]  R[157] mm/sec FINE Offset,PR[76:Offst_dprt] ;
2912:L P[1926]  R[157] mm/sec CNT100 Offset,PR[24:Rotate_Offset] ;
2913:L P[1927]  R[157] mm/sec CNT100 Offset,PR[24:Rotate_Offset] ;
2914:L P[1928]  R[157] mm/sec CNT100 Offset,PR[24:Rotate_Offset] ;
2915:L P[1929]  R[157] mm/sec CNT100 Offset,PR[24:Rotate_Offset] ;
2916:L P[1930]  R[157] mm/sec CNT100 Offset,PR[24:Rotate_Offset] ;
2917:L P[1931]  R[157] mm/sec CNT100 Offset,PR[24:Rotate_Offset] ;
2918: !Pass140 ;
2919: LBL[1140:Pass140] ;
2920:L P[1932]  R[157] mm/sec FINE Offset,PR[78:Offst_apprch]  ;
2921: WAIT   0.20(sec) ;
2922:L P[1932]  R[157] mm/sec CNT100 TA    0.00sec,CALL RUN_LASER_START Offset,PR[25:Start_Offset] ;
2924:L P[1933]  R[157] mm/sec CNT100 Offset,PR[24:Rotate_Offset] ;
2925:L P[1934]  R[157] mm/sec CNT100 TA    0.00sec,CALL RUN_LASER_STOP Offset,PR[26:Stop_Offset] ;
2927:L P[1934]  R[157] mm/sec FINE Offset,PR[76:Offst_dprt] ;
2928:L P[1935]  R[157] mm/sec CNT100 Offset,PR[24:Rotate_Offset] ;
2929:L P[1936]  R[157] mm/sec CNT100 Offset,PR[24:Rotate_Offset] ;
2930:L P[1937]  R[157] mm/sec CNT100 Offset,PR[24:Rotate_Offset] ;
2931:L P[1938]  R[157] mm/sec CNT100 Offset,PR[24:Rotate_Offset] ;
2932:L P[1939]  R[157] mm/sec CNT100 Offset,PR[24:Rotate_Offset] ;
2933:L P[1940]  R[157] mm/sec CNT100 Offset,PR[24:Rotate_Offset] ;
2934: !Pass141 ;
2935: LBL[1141:Pass141] ;
2936:L P[1941]  R[157] mm/sec FINE Offset,PR[78:Offst_apprch]  ;
2937: WAIT   0.20(sec) ;
2938:L P[1941]  R[157] mm/sec CNT100 TA    0.00sec,CALL RUN_LASER_START Offset,PR[25:Start_Offset] ;
2940:L P[1942]  R[157] mm/sec CNT100 Offset,PR[24:Rotate_Offset] ;
2941:L P[1943]  R[157] mm/sec CNT100 Offset,PR[24:Rotate_Offset] ;
2942:L P[1944]  R[157] mm/sec CNT100 Offset,PR[24:Rotate_Offset] ;
2943:L P[1945]  R[157] mm/sec CNT100 Offset,PR[24:Rotate_Offset] ;
2944:L P[1946]  R[157] mm/sec CNT100 Offset,PR[24:Rotate_Offset] ;
2945:L P[1947]  R[157] mm/sec CNT100 TA    0.00sec,CALL RUN_LASER_STOP Offset,PR[26:Stop_Offset] ;
2947:L P[1947]  R[157] mm/sec FINE Offset,PR[76:Offst_dprt] ;
2948:L P[1948]  R[157] mm/sec CNT100 Offset,PR[24:Rotate_Offset] ;
2949:L P[1949]  R[157] mm/sec CNT100 Offset,PR[24:Rotate_Offset] ;
2950:L P[1950]  R[157] mm/sec CNT100 Offset,PR[24:Rotate_Offset] ;
2951:L P[1951]  R[157] mm/sec CNT100 Offset,PR[24:Rotate_Offset] ;
2952:L P[1952]  R[157] mm/sec CNT100 Offset,PR[24:Rotate_Offset] ;
2953:L P[1953]  R[157] mm/sec CNT100 Offset,PR[24:Rotate_Offset] ;
2954: !Pass142 ;
2955: LBL[1142:Pass142] ;
2956:L P[1954]  R[157] mm/sec FINE Offset,PR[78:Offst_apprch]  ;
2957: WAIT   0.20(sec) ;
2958:L P[1954]  R[157] mm/sec CNT100 TA    0.00sec,CALL RUN_LASER_START Offset,PR[25:Start_Offset] ;
2960:L P[1955]  R[157] mm/sec CNT100 Offset,PR[24:Rotate_Offset] ;
2961:L P[1956]  R[157] mm/sec CNT100 Offset,PR[24:Rotate_Offset] ;
2962:L P[1957]  R[157] mm/sec CNT100 Offset,PR[24:Rotate_Offset] ;
2963:L P[1958]  R[157] mm/sec CNT100 TA    0.00sec,CALL RUN_LASER_STOP Offset,PR[26:Stop_Offset] ;
2965:L P[1958]  R[157] mm/sec FINE Offset,PR[76:Offst_dprt] ;
2966:L P[1959]  R[157] mm/sec CNT100 Offset,PR[24:Rotate_Offset] ;
2967:L P[1960]  R[157] mm/sec CNT100 Offset,PR[24:Rotate_Offset] ;
2968:L P[1961]  R[157] mm/sec CNT100 Offset,PR[24:Rotate_Offset] ;
2969:L P[1962]  R[157] mm/sec CNT100 Offset,PR[24:Rotate_Offset] ;
2970:L P[1963]  R[157] mm/sec CNT100 Offset,PR[24:Rotate_Offset] ;
2971:L P[1964]  R[157] mm/sec CNT100 Offset,PR[24:Rotate_Offset] ;
2972: !Pass143 ;
2973: LBL[1143:Pass143] ;
2974:L P[1965]  R[157] mm/sec FINE Offset,PR[78:Offst_apprch]  ;
2975: WAIT   0.20(sec) ;
2976:L P[1965]  R[157] mm/sec CNT100 TA    0.00sec,CALL RUN_LASER_START Offset,PR[25:Start_Offset] ;
2978:L P[1966]  R[157] mm/sec CNT100 Offset,PR[24:Rotate_Offset] ;
2979:L P[1967]  R[157] mm/sec CNT100 Offset,PR[24:Rotate_Offset] ;
2980:L P[1968]  R[157] mm/sec CNT100 Offset,PR[24:Rotate_Offset] ;
2981:L P[1969]  R[157] mm/sec CNT100 TA    0.00sec,CALL RUN_LASER_STOP Offset,PR[26:Stop_Offset] ;
2983:L P[1969]  R[157] mm/sec FINE Offset,PR[76:Offst_dprt] ;
2984:L P[1970]  R[157] mm/sec CNT100 Offset,PR[24:Rotate_Offset] ;
2985:L P[1971]  R[157] mm/sec CNT100 Offset,PR[24:Rotate_Offset] ;
2986:L P[1972]  R[157] mm/sec CNT100 Offset,PR[24:Rotate_Offset] ;
2987:L P[1973]  R[157] mm/sec CNT100 Offset,PR[24:Rotate_Offset] ;
2988:L P[1974]  R[157] mm/sec CNT100 Offset,PR[24:Rotate_Offset] ;
2989:L P[1975]  R[157] mm/sec CNT100 Offset,PR[24:Rotate_Offset] ;
2990: !Pass144 ;
2991: LBL[1144:Pass144] ;
2992:L P[1976]  R[157] mm/sec FINE Offset,PR[78:Offst_apprch]  ;
2993: WAIT   0.20(sec) ;
2994:L P[1976]  R[157] mm/sec CNT100 TA    0.00sec,CALL RUN_LASER_START Offset,PR[25:Start_Offset] ;
2996:L P[1977]  R[157] mm/sec CNT100 Offset,PR[24:Rotate_Offset] ;
2997:L P[1978]  R[157] mm/sec CNT100 Offset,PR[24:Rotate_Offset] ;
2998:L P[1979]  R[157] mm/sec CNT100 Offset,PR[24:Rotate_Offset] ;
2999:L P[1980]  R[157] mm/sec CNT100 TA    0.00sec,CALL RUN_LASER_STOP Offset,PR[26:Stop_Offset] ;
3001:L P[1980]  R[157] mm/sec FINE Offset,PR[76:Offst_dprt] ;
3002:L P[1981]  R[157] mm/sec CNT100 Offset,PR[24:Rotate_Offset] ;
3003:L P[1982]  R[157] mm/sec CNT100 Offset,PR[24:Rotate_Offset] ;
3004:L P[1983]  R[157] mm/sec CNT100 Offset,PR[24:Rotate_Offset] ;
3005:L P[1984]  R[157] mm/sec CNT100 Offset,PR[24:Rotate_Offset] ;
3006:L P[1985]  R[157] mm/sec CNT100 Offset,PR[24:Rotate_Offset] ;
3007:L P[1986]  R[157] mm/sec CNT100 Offset,PR[24:Rotate_Offset] ;
3008: !Pass145 ;
3009: LBL[1145:Pass145] ;
3010:L P[1987]  R[157] mm/sec FINE Offset,PR[78:Offst_apprch]  ;
3011: WAIT   0.20(sec) ;
3012:L P[1987]  R[157] mm/sec CNT100 TA    0.00sec,CALL RUN_LASER_START Offset,PR[25:Start_Offset] ;
3014:L P[1988]  R[157] mm/sec CNT100 Offset,PR[24:Rotate_Offset] ;
3015:L P[1989]  R[157] mm/sec CNT100 Offset,PR[24:Rotate_Offset] ;
3016:L P[1990]  R[157] mm/sec CNT100 Offset,PR[24:Rotate_Offset] ;
3017:L P[1991]  R[157] mm/sec CNT100 TA    0.00sec,CALL RUN_LASER_STOP Offset,PR[26:Stop_Offset] ;
3019:L P[1991]  R[157] mm/sec FINE Offset,PR[76:Offst_dprt] ;
3020:L P[1992]  R[157] mm/sec CNT100 Offset,PR[24:Rotate_Offset] ;
3021:L P[1993]  R[157] mm/sec CNT100 Offset,PR[24:Rotate_Offset] ;
3022:L P[1994]  R[157] mm/sec CNT100 Offset,PR[24:Rotate_Offset] ;
3023:L P[1995]  R[157] mm/sec CNT100 Offset,PR[24:Rotate_Offset] ;
3024:L P[1996]  R[157] mm/sec CNT100 Offset,PR[24:Rotate_Offset] ;
3025:L P[1997]  R[157] mm/sec CNT100 Offset,PR[24:Rotate_Offset] ;
3026: !Pass146 ;
3027: LBL[1146:Pass146] ;
3028:L P[1998]  R[157] mm/sec FINE Offset,PR[78:Offst_apprch]  ;
3029: WAIT   0.20(sec) ;
3030:L P[1998]  R[157] mm/sec CNT100 TA    0.00sec,CALL RUN_LASER_START Offset,PR[25:Start_Offset] ;
3032:L P[1999]  R[157] mm/sec CNT100 Offset,PR[24:Rotate_Offset] ;
3033:L P[2000]  R[157] mm/sec CNT100 Offset,PR[24:Rotate_Offset] ;
3034:L P[2001]  R[157] mm/sec CNT100 Offset,PR[24:Rotate_Offset] ;
3035:L P[2002]  R[157] mm/sec CNT100 TA    0.00sec,CALL RUN_LASER_STOP Offset,PR[26:Stop_Offset] ;
3037:L P[2002]  R[157] mm/sec FINE Offset,PR[76:Offst_dprt] ;
3038:L P[2003]  R[157] mm/sec CNT100 Offset,PR[24:Rotate_Offset] ;
3039:L P[2004]  R[157] mm/sec CNT100 Offset,PR[24:Rotate_Offset] ;
3040:L P[2005]  R[157] mm/sec CNT100 Offset,PR[24:Rotate_Offset] ;
3041:L P[2006]  R[157] mm/sec CNT100 Offset,PR[24:Rotate_Offset] ;
3042:L P[2007]  R[157] mm/sec CNT100 Offset,PR[24:Rotate_Offset] ;
3043:L P[2008]  R[157] mm/sec CNT100 Offset,PR[24:Rotate_Offset] ;
3044: !Pass147 ;
3045: LBL[1147:Pass147] ;
3046:L P[2009]  R[157] mm/sec FINE Offset,PR[78:Offst_apprch]  ;
3047: WAIT   0.20(sec) ;
3048:L P[2009]  R[157] mm/sec CNT100 TA    0.00sec,CALL RUN_LASER_START Offset,PR[25:Start_Offset] ;
3050:L P[2010]  R[157] mm/sec CNT100 Offset,PR[24:Rotate_Offset] ;
3051:L P[2011]  R[157] mm/sec CNT100 TA    0.00sec,CALL RUN_LASER_STOP Offset,PR[26:Stop_Offset] ;
3053:L P[2011]  R[157] mm/sec FINE Offset,PR[76:Offst_dprt] ;
3054:L P[2012]  R[157] mm/sec CNT100 Offset,PR[24:Rotate_Offset] ;
3055:L P[2013]  R[157] mm/sec CNT100 Offset,PR[24:Rotate_Offset] ;
3056:L P[2014]  R[157] mm/sec CNT100 Offset,PR[24:Rotate_Offset] ;
3057:L P[2015]  R[157] mm/sec CNT100 Offset,PR[24:Rotate_Offset] ;
3058:L P[2016]  R[157] mm/sec CNT100 Offset,PR[24:Rotate_Offset] ;
3059:L P[2017]  R[157] mm/sec CNT100 Offset,PR[24:Rotate_Offset] ;
3060: !Pass148 ;
3061: LBL[1148:Pass148] ;
3062:L P[2018]  R[157] mm/sec FINE Offset,PR[78:Offst_apprch]  ;
3063: WAIT   0.20(sec) ;
3064:L P[2018]  R[157] mm/sec CNT100 TA    0.00sec,CALL RUN_LASER_START Offset,PR[25:Start_Offset] ;
3066:L P[2019]  R[157] mm/sec CNT100 Offset,PR[24:Rotate_Offset] ;
3067:L P[2020]  R[157] mm/sec CNT100 TA    0.00sec,CALL RUN_LASER_STOP Offset,PR[26:Stop_Offset] ;
3069:L P[2020]  R[157] mm/sec FINE Offset,PR[76:Offst_dprt] ;
3070:L P[2021]  R[157] mm/sec CNT100 Offset,PR[24:Rotate_Offset] ;
3071:L P[2022]  R[157] mm/sec CNT100 Offset,PR[24:Rotate_Offset] ;
3072:L P[2023]  R[157] mm/sec CNT100 Offset,PR[24:Rotate_Offset] ;
3073:L P[2024]  R[157] mm/sec CNT100 Offset,PR[24:Rotate_Offset] ;
3074:L P[2025]  R[157] mm/sec CNT100 Offset,PR[24:Rotate_Offset] ;
3075:L P[2026]  R[157] mm/sec CNT100 Offset,PR[24:Rotate_Offset] ;
3076: !Pass149 ;
3077: LBL[1149:Pass149] ;
3078:L P[2027]  R[157] mm/sec FINE Offset,PR[78:Offst_apprch]  ;
3079: WAIT   0.20(sec) ;
3080:L P[2027]  R[157] mm/sec CNT100 TA    0.00sec,CALL RUN_LASER_START Offset,PR[25:Start_Offset] ;
3082:L P[2028]  R[157] mm/sec CNT100 Offset,PR[24:Rotate_Offset] ;
3083:L P[2029]  R[157] mm/sec CNT100 Offset,PR[24:Rotate_Offset] ;
3084:L P[2030]  R[157] mm/sec CNT100 Offset,PR[24:Rotate_Offset] ;
3085:L P[2031]  R[157] mm/sec CNT100 TA    0.00sec,CALL RUN_LASER_STOP Offset,PR[26:Stop_Offset] ;
3087:L P[2031]  R[157] mm/sec FINE Offset,PR[76:Offst_dprt] ;
3088:L P[2032]  R[157] mm/sec CNT100 Offset,PR[24:Rotate_Offset] ;
3089:L P[2033]  R[157] mm/sec CNT100 Offset,PR[24:Rotate_Offset] ;
3090:L P[2034]  R[157] mm/sec CNT100 Offset,PR[24:Rotate_Offset] ;
3091:L P[2035]  R[157] mm/sec CNT100 Offset,PR[24:Rotate_Offset] ;
3092:L P[2036]  R[157] mm/sec CNT100 Offset,PR[24:Rotate_Offset] ;
3093:L P[2037]  R[157] mm/sec CNT100 Offset,PR[24:Rotate_Offset] ;
3094: !Pass150 ;
3095: LBL[1150:Pass150] ;
3096:L P[2038]  R[157] mm/sec FINE Offset,PR[78:Offst_apprch]  ;
3097: WAIT   0.20(sec) ;
3098:L P[2038]  R[157] mm/sec CNT100 TA    0.00sec,CALL RUN_LASER_START Offset,PR[25:Start_Offset] ;
3100:L P[2039]  R[157] mm/sec CNT100 Offset,PR[24:Rotate_Offset] ;
3101:L P[2040]  R[157] mm/sec CNT100 Offset,PR[24:Rotate_Offset] ;
3102:L P[2041]  R[157] mm/sec CNT100 Offset,PR[24:Rotate_Offset] ;
3103:L P[2042]  R[157] mm/sec CNT100 TA    0.00sec,CALL RUN_LASER_STOP Offset,PR[26:Stop_Offset] ;
3105:L P[2042]  R[157] mm/sec FINE Offset,PR[76:Offst_dprt] ;
3106:L P[2043]  R[157] mm/sec CNT100 Offset,PR[24:Rotate_Offset] ;
3107:L P[2044]  R[157] mm/sec CNT100 Offset,PR[24:Rotate_Offset] ;
3108:L P[2045]  R[157] mm/sec CNT100 Offset,PR[24:Rotate_Offset] ;
3109:L P[2046]  R[157] mm/sec CNT100 Offset,PR[24:Rotate_Offset] ;
3110:L P[2047]  R[157] mm/sec CNT100 Offset,PR[24:Rotate_Offset] ;
3111:L P[2048]  R[157] mm/sec CNT100 Offset,PR[24:Rotate_Offset] ;
3112: !Pass151 ;
3113: LBL[1151:Pass151] ;
3114:L P[2049]  R[157] mm/sec FINE Offset,PR[78:Offst_apprch]  ;
3115: WAIT   0.20(sec) ;
3116:L P[2049]  R[157] mm/sec CNT100 TA    0.00sec,CALL RUN_LASER_START Offset,PR[25:Start_Offset] ;
3118:L P[2050]  R[157] mm/sec CNT100 Offset,PR[24:Rotate_Offset] ;
3119:L P[2051]  R[157] mm/sec CNT100 Offset,PR[24:Rotate_Offset] ;
3120:L P[2052]  R[157] mm/sec CNT100 Offset,PR[24:Rotate_Offset] ;
3121:L P[2053]  R[157] mm/sec CNT100 TA    0.00sec,CALL RUN_LASER_STOP Offset,PR[26:Stop_Offset] ;
3123:L P[2053]  R[157] mm/sec FINE Offset,PR[76:Offst_dprt] ;
3124:L P[2054]  R[157] mm/sec CNT100 Offset,PR[24:Rotate_Offset] ;
3125:L P[2055]  R[157] mm/sec CNT100 Offset,PR[24:Rotate_Offset] ;
3126:L P[2056]  R[157] mm/sec CNT100 Offset,PR[24:Rotate_Offset] ;
3127:L P[2057]  R[157] mm/sec CNT100 Offset,PR[24:Rotate_Offset] ;
3128:L P[2058]  R[157] mm/sec CNT100 Offset,PR[24:Rotate_Offset] ;
3129:L P[2059]  R[157] mm/sec CNT100 Offset,PR[24:Rotate_Offset] ;
3130: !Pass152 ;
3131: LBL[1152:Pass152] ;
3132:L P[2060]  R[157] mm/sec FINE Offset,PR[78:Offst_apprch]  ;
3133: WAIT   0.20(sec) ;
3134:L P[2060]  R[157] mm/sec CNT100 TA    0.00sec,CALL RUN_LASER_START Offset,PR[25:Start_Offset] ;
3136:L P[2061]  R[157] mm/sec CNT100 Offset,PR[24:Rotate_Offset] ;
3137:L P[2062]  R[157] mm/sec CNT100 Offset,PR[24:Rotate_Offset] ;
3138:L P[2063]  R[157] mm/sec CNT100 Offset,PR[24:Rotate_Offset] ;
3139:L P[2064]  R[157] mm/sec CNT100 TA    0.00sec,CALL RUN_LASER_STOP Offset,PR[26:Stop_Offset] ;
3141:L P[2064]  R[157] mm/sec FINE Offset,PR[76:Offst_dprt] ;
3142:L P[2065]  R[157] mm/sec CNT100 Offset,PR[24:Rotate_Offset] ;
3143:L P[2066]  R[157] mm/sec CNT100 Offset,PR[24:Rotate_Offset] ;
3144:L P[2067]  R[157] mm/sec CNT100 Offset,PR[24:Rotate_Offset] ;
3145:L P[2068]  R[157] mm/sec CNT100 Offset,PR[24:Rotate_Offset] ;
3146:L P[2069]  R[157] mm/sec CNT100 Offset,PR[24:Rotate_Offset] ;
3147:L P[2070]  R[157] mm/sec CNT100 Offset,PR[24:Rotate_Offset] ;
3148: !Pass153 ;
3149: LBL[1153:Pass153] ;
3150:L P[2071]  R[157] mm/sec FINE Offset,PR[78:Offst_apprch]  ;
3151: WAIT   0.20(sec) ;
3152:L P[2071]  R[157] mm/sec CNT100 TA    0.00sec,CALL RUN_LASER_START Offset,PR[25:Start_Offset] ;
3154:L P[2072]  R[157] mm/sec CNT100 Offset,PR[24:Rotate_Offset] ;
3155:L P[2073]  R[157] mm/sec CNT100 Offset,PR[24:Rotate_Offset] ;
3156:L P[2074]  R[157] mm/sec CNT100 Offset,PR[24:Rotate_Offset] ;
3157:L P[2075]  R[157] mm/sec CNT100 TA    0.00sec,CALL RUN_LASER_STOP Offset,PR[26:Stop_Offset] ;
3159:L P[2075]  R[157] mm/sec FINE Offset,PR[76:Offst_dprt] ;
3160:L P[2076]  R[157] mm/sec CNT100 Offset,PR[24:Rotate_Offset] ;
3161:L P[2077]  R[157] mm/sec CNT100 Offset,PR[24:Rotate_Offset] ;
3162:L P[2078]  R[157] mm/sec CNT100 Offset,PR[24:Rotate_Offset] ;
3163:L P[2079]  R[157] mm/sec CNT100 Offset,PR[24:Rotate_Offset] ;
3164:L P[2080]  R[157] mm/sec CNT100 Offset,PR[24:Rotate_Offset] ;
3165:L P[2081]  R[157] mm/sec CNT100 Offset,PR[24:Rotate_Offset] ;
3166: !Pass154 ;
3167: LBL[1154:Pass154] ;
3168:L P[2082]  R[157] mm/sec FINE Offset,PR[78:Offst_apprch]  ;
3169: WAIT   0.20(sec) ;
3170:L P[2082]  R[157] mm/sec CNT100 TA    0.00sec,CALL RUN_LASER_START Offset,PR[25:Start_Offset] ;
3172:L P[2083]  R[157] mm/sec CNT100 Offset,PR[24:Rotate_Offset] ;
3173:L P[2084]  R[157] mm/sec CNT100 Offset,PR[24:Rotate_Offset] ;
3174:L P[2085]  R[157] mm/sec CNT100 Offset,PR[24:Rotate_Offset] ;
3175:L P[2086]  R[157] mm/sec CNT100 Offset,PR[24:Rotate_Offset] ;
3176:L P[2087]  R[157] mm/sec CNT100 Offset,PR[24:Rotate_Offset] ;
3177:L P[2088]  R[157] mm/sec CNT100 Offset,PR[24:Rotate_Offset] ;
3178:L P[2089]  R[157] mm/sec CNT100 TA    0.00sec,CALL RUN_LASER_STOP Offset,PR[26:Stop_Offset] ;
3180:L P[2089]  R[157] mm/sec FINE Offset,PR[76:Offst_dprt] ;
3181:L P[2090]  R[157] mm/sec CNT100 Offset,PR[24:Rotate_Offset] ;
3182:L P[2091]  R[157] mm/sec CNT100 Offset,PR[24:Rotate_Offset] ;
3183:L P[2092]  R[157] mm/sec CNT100 Offset,PR[24:Rotate_Offset] ;
3184:L P[2093]  R[157] mm/sec CNT100 Offset,PR[24:Rotate_Offset] ;
3185:L P[2094]  R[157] mm/sec CNT100 Offset,PR[24:Rotate_Offset] ;
3186:L P[2095]  R[157] mm/sec CNT100 Offset,PR[24:Rotate_Offset] ;
3187: !Pass155 ;
3188: LBL[1155:Pass155] ;
3189:L P[2096]  R[157] mm/sec FINE Offset,PR[78:Offst_apprch]  ;
3190: WAIT   0.20(sec) ;
3191:L P[2096]  R[157] mm/sec CNT100 TA    0.00sec,CALL RUN_LASER_START Offset,PR[25:Start_Offset] ;
3193:L P[2097]  R[157] mm/sec CNT100 Offset,PR[24:Rotate_Offset] ;
3194:L P[2098]  R[157] mm/sec CNT100 TA    0.00sec,CALL RUN_LASER_STOP Offset,PR[26:Stop_Offset] ;
3196:L P[2098]  R[157] mm/sec FINE Offset,PR[76:Offst_dprt] ;
3197:L P[2099]  R[157] mm/sec CNT100 Offset,PR[24:Rotate_Offset] ;
3198:L P[2100]  R[157] mm/sec CNT100 Offset,PR[24:Rotate_Offset] ;
3199:L P[2101]  R[157] mm/sec CNT100 Offset,PR[24:Rotate_Offset] ;
3200:L P[2102]  R[157] mm/sec CNT100 Offset,PR[24:Rotate_Offset] ;
3201:L P[2103]  R[157] mm/sec CNT100 Offset,PR[24:Rotate_Offset] ;
3202:L P[2104]  R[157] mm/sec CNT100 Offset,PR[24:Rotate_Offset] ;
3203: !Pass156 ;
3204: LBL[1156:Pass156] ;
3205:L P[2105]  R[157] mm/sec FINE Offset,PR[78:Offst_apprch]  ;
3206: WAIT   0.20(sec) ;
3207:L P[2105]  R[157] mm/sec CNT100 TA    0.00sec,CALL RUN_LASER_START Offset,PR[25:Start_Offset] ;
3209:L P[2106]  R[157] mm/sec CNT100 Offset,PR[24:Rotate_Offset] ;
3210:L P[2107]  R[157] mm/sec CNT100 TA    0.00sec,CALL RUN_LASER_STOP Offset,PR[26:Stop_Offset] ;
3212:L P[2107]  R[157] mm/sec FINE Offset,PR[76:Offst_dprt] ;
3213:L P[2108]  R[157] mm/sec CNT100 Offset,PR[24:Rotate_Offset] ;
3214:L P[2109]  R[157] mm/sec CNT100 Offset,PR[24:Rotate_Offset] ;
3215:L P[2110]  R[157] mm/sec CNT100 Offset,PR[24:Rotate_Offset] ;
3216:L P[2111]  R[157] mm/sec CNT100 Offset,PR[24:Rotate_Offset] ;
3217:L P[2112]  R[157] mm/sec CNT100 Offset,PR[24:Rotate_Offset] ;
3218:L P[2113]  R[157] mm/sec CNT100 Offset,PR[24:Rotate_Offset] ;
3219: !Pass157 ;
3220: LBL[1157:Pass157] ;
3221:L P[2114]  R[157] mm/sec FINE Offset,PR[78:Offst_apprch]  ;
3222: WAIT   0.20(sec) ;
3223:L P[2114]  R[157] mm/sec CNT100 TA    0.00sec,CALL RUN_LASER_START Offset,PR[25:Start_Offset] ;
3225:L P[2115]  R[157] mm/sec CNT100 Offset,PR[24:Rotate_Offset] ;
3226:L P[2116]  R[157] mm/sec CNT100 Offset,PR[24:Rotate_Offset] ;
3227:L P[2117]  R[157] mm/sec CNT100 Offset,PR[24:Rotate_Offset] ;
3228:L P[2118]  R[157] mm/sec CNT100 Offset,PR[24:Rotate_Offset] ;
3229:L P[2119]  R[157] mm/sec CNT100 Offset,PR[24:Rotate_Offset] ;
3230:L P[2120]  R[157] mm/sec CNT100 TA    0.00sec,CALL RUN_LASER_STOP Offset,PR[26:Stop_Offset] ;
3232:L P[2120]  R[157] mm/sec FINE Offset,PR[76:Offst_dprt] ;
3233:L P[2121]  R[157] mm/sec CNT100 Offset,PR[24:Rotate_Offset] ;
3234:L P[2122]  R[157] mm/sec CNT100 Offset,PR[24:Rotate_Offset] ;
3235:L P[2123]  R[157] mm/sec CNT100 Offset,PR[24:Rotate_Offset] ;
3236:L P[2124]  R[157] mm/sec CNT100 Offset,PR[24:Rotate_Offset] ;
3237:L P[2125]  R[157] mm/sec CNT100 Offset,PR[24:Rotate_Offset] ;
3238:L P[2126]  R[157] mm/sec CNT100 Offset,PR[24:Rotate_Offset] ;
3239: !Pass158 ;
3240: LBL[1158:Pass158] ;
3241:L P[2127]  R[157] mm/sec FINE Offset,PR[78:Offst_apprch]  ;
3242: WAIT   0.20(sec) ;
3243:L P[2127]  R[157] mm/sec CNT100 TA    0.00sec,CALL RUN_LASER_START Offset,PR[25:Start_Offset] ;
3245:L P[2128]  R[157] mm/sec CNT100 Offset,PR[24:Rotate_Offset] ;
3246:L P[2129]  R[157] mm/sec CNT100 Offset,PR[24:Rotate_Offset] ;
3247:L P[2130]  R[157] mm/sec CNT100 Offset,PR[24:Rotate_Offset] ;
3248:L P[2131]  R[157] mm/sec CNT100 TA    0.00sec,CALL RUN_LASER_STOP Offset,PR[26:Stop_Offset] ;
3250:L P[2131]  R[157] mm/sec FINE Offset,PR[76:Offst_dprt] ;
3251:L P[2132]  R[157] mm/sec CNT100 Offset,PR[24:Rotate_Offset] ;
3252:L P[2133]  R[157] mm/sec CNT100 Offset,PR[24:Rotate_Offset] ;
3253:L P[2134]  R[157] mm/sec CNT100 Offset,PR[24:Rotate_Offset] ;
3254:L P[2135]  R[157] mm/sec CNT100 Offset,PR[24:Rotate_Offset] ;
3255:L P[2136]  R[157] mm/sec CNT100 Offset,PR[24:Rotate_Offset] ;
3256:L P[2137]  R[157] mm/sec CNT100 Offset,PR[24:Rotate_Offset] ;
3257: !Pass159 ;
3258: LBL[1159:Pass159] ;
3259:L P[2138]  R[157] mm/sec FINE Offset,PR[78:Offst_apprch]  ;
3260: WAIT   0.20(sec) ;
3261:L P[2138]  R[157] mm/sec CNT100 TA    0.00sec,CALL RUN_LASER_START Offset,PR[25:Start_Offset] ;
3263:L P[2139]  R[157] mm/sec CNT100 Offset,PR[24:Rotate_Offset] ;
3264:L P[2140]  R[157] mm/sec CNT100 Offset,PR[24:Rotate_Offset] ;
3265:L P[2141]  R[157] mm/sec CNT100 TA    0.00sec,CALL RUN_LASER_STOP Offset,PR[26:Stop_Offset] ;
3267:L P[2141]  R[157] mm/sec FINE Offset,PR[76:Offst_dprt] ;
3268:L P[2142]  R[157] mm/sec CNT100 Offset,PR[24:Rotate_Offset] ;
3269:L P[2143]  R[157] mm/sec CNT100 Offset,PR[24:Rotate_Offset] ;
3270:L P[2144]  R[157] mm/sec CNT100 Offset,PR[24:Rotate_Offset] ;
3271:L P[2145]  R[157] mm/sec CNT100 Offset,PR[24:Rotate_Offset] ;
3272:L P[2146]  R[157] mm/sec CNT100 Offset,PR[24:Rotate_Offset] ;
3273:L P[2147]  R[157] mm/sec CNT100 Offset,PR[24:Rotate_Offset] ;
3274: !Pass160 ;
3275: LBL[1160:Pass160] ;
3276:L P[2148]  R[157] mm/sec FINE Offset,PR[78:Offst_apprch]  ;
3277: WAIT   0.20(sec) ;
3278:L P[2148]  R[157] mm/sec CNT100 TA    0.00sec,CALL RUN_LASER_START Offset,PR[25:Start_Offset] ;
3280:L P[2149]  R[157] mm/sec CNT100 Offset,PR[24:Rotate_Offset] ;
3281:L P[2150]  R[157] mm/sec CNT100 Offset,PR[24:Rotate_Offset] ;
3282:L P[2151]  R[157] mm/sec CNT100 TA    0.00sec,CALL RUN_LASER_STOP Offset,PR[26:Stop_Offset] ;
3284:L P[2151]  R[157] mm/sec FINE Offset,PR[76:Offst_dprt] ;
3285:L P[2152]  R[157] mm/sec CNT100 Offset,PR[24:Rotate_Offset] ;
3286:L P[2153]  R[157] mm/sec CNT100 Offset,PR[24:Rotate_Offset] ;
3287:L P[2154]  R[157] mm/sec CNT100 Offset,PR[24:Rotate_Offset] ;
3288:L P[2155]  R[157] mm/sec CNT100 Offset,PR[24:Rotate_Offset] ;
3289:L P[2156]  R[157] mm/sec CNT100 Offset,PR[24:Rotate_Offset] ;
3290:L P[2157]  R[157] mm/sec CNT100 Offset,PR[24:Rotate_Offset] ;
3291: !Pass161 ;
3292: LBL[1161:Pass161] ;
3293:L P[2158]  R[157] mm/sec FINE Offset,PR[78:Offst_apprch]  ;
3294: WAIT   0.20(sec) ;
3295:L P[2158]  R[157] mm/sec CNT100 TA    0.00sec,CALL RUN_LASER_START Offset,PR[25:Start_Offset] ;
3297:L P[2159]  R[157] mm/sec CNT100 Offset,PR[24:Rotate_Offset] ;
3298:L P[2160]  R[157] mm/sec CNT100 Offset,PR[24:Rotate_Offset] ;
3299:L P[2161]  R[157] mm/sec CNT100 Offset,PR[24:Rotate_Offset] ;
3300:L P[2162]  R[157] mm/sec CNT100 TA    0.00sec,CALL RUN_LASER_STOP Offset,PR[26:Stop_Offset] ;
3302:L P[2162]  R[157] mm/sec FINE Offset,PR[76:Offst_dprt] ;
3303:L P[2163]  R[157] mm/sec CNT100 Offset,PR[24:Rotate_Offset] ;
3304:L P[2164]  R[157] mm/sec CNT100 Offset,PR[24:Rotate_Offset] ;
3305:L P[2165]  R[157] mm/sec CNT100 Offset,PR[24:Rotate_Offset] ;
3306:L P[2166]  R[157] mm/sec CNT100 Offset,PR[24:Rotate_Offset] ;
3307:L P[2167]  R[157] mm/sec CNT100 Offset,PR[24:Rotate_Offset] ;
3308:L P[2168]  R[157] mm/sec CNT100 Offset,PR[24:Rotate_Offset] ;
3309: !Pass162 ;
3310: LBL[1162:Pass162] ;
3311:L P[2169]  R[157] mm/sec FINE Offset,PR[78:Offst_apprch]  ;
3312: WAIT   0.20(sec) ;
3313:L P[2169]  R[157] mm/sec CNT100 TA    0.00sec,CALL RUN_LASER_START Offset,PR[25:Start_Offset] ;
3315:L P[2170]  R[157] mm/sec CNT100 Offset,PR[24:Rotate_Offset] ;
3316:L P[2171]  R[157] mm/sec CNT100 Offset,PR[24:Rotate_Offset] ;
3317:L P[2172]  R[157] mm/sec CNT100 Offset,PR[24:Rotate_Offset] ;
3318:L P[2173]  R[157] mm/sec CNT100 TA    0.00sec,CALL RUN_LASER_STOP Offset,PR[26:Stop_Offset] ;
3320:L P[2173]  R[157] mm/sec FINE Offset,PR[76:Offst_dprt] ;
3321:L P[2174]  R[157] mm/sec CNT100 Offset,PR[24:Rotate_Offset] ;
3322:L P[2175]  R[157] mm/sec CNT100 Offset,PR[24:Rotate_Offset] ;
3323:L P[2176]  R[157] mm/sec CNT100 Offset,PR[24:Rotate_Offset] ;
3324:L P[2177]  R[157] mm/sec CNT100 Offset,PR[24:Rotate_Offset] ;
3325:L P[2178]  R[157] mm/sec CNT100 Offset,PR[24:Rotate_Offset] ;
3326:L P[2179]  R[157] mm/sec CNT100 Offset,PR[24:Rotate_Offset] ;
3327: !Pass163 ;
3328: LBL[1163:Pass163] ;
3329:L P[2180]  R[157] mm/sec FINE Offset,PR[78:Offst_apprch]  ;
3330: WAIT   0.20(sec) ;
3331:L P[2180]  R[157] mm/sec CNT100 TA    0.00sec,CALL RUN_LASER_START Offset,PR[25:Start_Offset] ;
3333:L P[2181]  R[157] mm/sec CNT100 Offset,PR[24:Rotate_Offset] ;
3334:L P[2182]  R[157] mm/sec CNT100 TA    0.00sec,CALL RUN_LASER_STOP Offset,PR[26:Stop_Offset] ;
3336:L P[2182]  R[157] mm/sec FINE Offset,PR[76:Offst_dprt] ;
3337:L P[2183]  R[157] mm/sec CNT100 Offset,PR[24:Rotate_Offset] ;
3338:L P[2184]  R[157] mm/sec CNT100 Offset,PR[24:Rotate_Offset] ;
3339:L P[2185]  R[157] mm/sec CNT100 Offset,PR[24:Rotate_Offset] ;
3340:L P[2186]  R[157] mm/sec CNT100 Offset,PR[24:Rotate_Offset] ;
3341:L P[2187]  R[157] mm/sec CNT100 Offset,PR[24:Rotate_Offset] ;
3342:L P[2188]  R[157] mm/sec CNT100 Offset,PR[24:Rotate_Offset] ;
3343: !Pass164 ;
3344: LBL[1164:Pass164] ;
3345:L P[2189]  R[157] mm/sec FINE Offset,PR[78:Offst_apprch]  ;
3346: WAIT   0.20(sec) ;
3347:L P[2189]  R[157] mm/sec CNT100 TA    0.00sec,CALL RUN_LASER_START Offset,PR[25:Start_Offset] ;
3349:L P[2190]  R[157] mm/sec CNT100 Offset,PR[24:Rotate_Offset] ;
3350:L P[2191]  R[157] mm/sec CNT100 TA    0.00sec,CALL RUN_LASER_STOP Offset,PR[26:Stop_Offset] ;
3352:L P[2191]  R[157] mm/sec FINE Offset,PR[76:Offst_dprt] ;
3353:L P[2192]  R[157] mm/sec CNT100 Offset,PR[24:Rotate_Offset] ;
3354:L P[2193]  R[157] mm/sec CNT100 Offset,PR[24:Rotate_Offset] ;
3355:L P[2194]  R[157] mm/sec CNT100 Offset,PR[24:Rotate_Offset] ;
3356:L P[2195]  R[157] mm/sec CNT100 Offset,PR[24:Rotate_Offset] ;
3357:L P[2196]  R[157] mm/sec CNT100 Offset,PR[24:Rotate_Offset] ;
3358:L P[2197]  R[157] mm/sec CNT100 Offset,PR[24:Rotate_Offset] ;
3359: !Pass165 ;
3360: LBL[1165:Pass165] ;
3361:L P[2198]  R[157] mm/sec FINE Offset,PR[78:Offst_apprch]  ;
3362: WAIT   0.20(sec) ;
3363:L P[2198]  R[157] mm/sec CNT100 TA    0.00sec,CALL RUN_LASER_START Offset,PR[25:Start_Offset] ;
3365:L P[2199]  R[157] mm/sec CNT100 Offset,PR[24:Rotate_Offset] ;
3366:L P[2200]  R[157] mm/sec CNT100 Offset,PR[24:Rotate_Offset] ;
3367:L P[2201]  R[157] mm/sec CNT100 Offset,PR[24:Rotate_Offset] ;
3368:L P[2202]  R[157] mm/sec CNT100 TA    0.00sec,CALL RUN_LASER_STOP Offset,PR[26:Stop_Offset] ;
3370:L P[2202]  R[157] mm/sec FINE Offset,PR[76:Offst_dprt] ;
3371:L P[2203]  R[157] mm/sec CNT100 Offset,PR[24:Rotate_Offset] ;
3372:L P[2204]  R[157] mm/sec CNT100 Offset,PR[24:Rotate_Offset] ;
3373:L P[2205]  R[157] mm/sec CNT100 Offset,PR[24:Rotate_Offset] ;
3374:L P[2206]  R[157] mm/sec CNT100 Offset,PR[24:Rotate_Offset] ;
3375:L P[2207]  R[157] mm/sec CNT100 Offset,PR[24:Rotate_Offset] ;
3376:L P[2208]  R[157] mm/sec CNT100 Offset,PR[24:Rotate_Offset] ;
3377: !Pass166 ;
3378: LBL[1166:Pass166] ;
3379:L P[2209]  R[157] mm/sec FINE Offset,PR[78:Offst_apprch]  ;
3380: WAIT   0.20(sec) ;
3381:L P[2209]  R[157] mm/sec CNT100 TA    0.00sec,CALL RUN_LASER_START Offset,PR[25:Start_Offset] ;
3383:L P[2210]  R[157] mm/sec CNT100 Offset,PR[24:Rotate_Offset] ;
3384:L P[2211]  R[157] mm/sec CNT100 Offset,PR[24:Rotate_Offset] ;
3385:L P[2212]  R[157] mm/sec CNT100 Offset,PR[24:Rotate_Offset] ;
3386:L P[2213]  R[157] mm/sec CNT100 TA    0.00sec,CALL RUN_LASER_STOP Offset,PR[26:Stop_Offset] ;
3388:L P[2213]  R[157] mm/sec FINE Offset,PR[76:Offst_dprt] ;
3389:L P[2214]  R[157] mm/sec CNT100 Offset,PR[24:Rotate_Offset] ;
3390:L P[2215]  R[157] mm/sec CNT100 Offset,PR[24:Rotate_Offset] ;
3391:L P[2216]  R[157] mm/sec CNT100 Offset,PR[24:Rotate_Offset] ;
3392:L P[2217]  R[157] mm/sec CNT100 Offset,PR[24:Rotate_Offset] ;
3393:L P[2218]  R[157] mm/sec CNT100 Offset,PR[24:Rotate_Offset] ;
3394:L P[2219]  R[157] mm/sec CNT100 Offset,PR[24:Rotate_Offset] ;
3395: !Pass167 ;
3396: LBL[1167:Pass167] ;
3397:L P[2220]  R[157] mm/sec FINE Offset,PR[78:Offst_apprch]  ;
3398: WAIT   0.20(sec) ;
3399:L P[2220]  R[157] mm/sec CNT100 TA    0.00sec,CALL RUN_LASER_START Offset,PR[25:Start_Offset] ;
3401:L P[2221]  R[157] mm/sec CNT100 Offset,PR[24:Rotate_Offset] ;
3402:L P[2222]  R[157] mm/sec CNT100 Offset,PR[24:Rotate_Offset] ;
3403:L P[2223]  R[157] mm/sec CNT100 Offset,PR[24:Rotate_Offset] ;
3404:L P[2224]  R[157] mm/sec CNT100 TA    0.00sec,CALL RUN_LASER_STOP Offset,PR[26:Stop_Offset] ;
3406:L P[2224]  R[157] mm/sec FINE Offset,PR[76:Offst_dprt] ;
3407:L P[2225]  R[157] mm/sec CNT100 Offset,PR[24:Rotate_Offset] ;
3408:L P[2226]  R[157] mm/sec CNT100 Offset,PR[24:Rotate_Offset] ;
3409:L P[2227]  R[157] mm/sec CNT100 Offset,PR[24:Rotate_Offset] ;
3410:L P[2228]  R[157] mm/sec CNT100 Offset,PR[24:Rotate_Offset] ;
3411:L P[2229]  R[157] mm/sec CNT100 Offset,PR[24:Rotate_Offset] ;
3412:L P[2230]  R[157] mm/sec CNT100 Offset,PR[24:Rotate_Offset] ;
3413: !Pass168 ;
3414: LBL[1168:Pass168] ;
3415:L P[2231]  R[157] mm/sec FINE Offset,PR[78:Offst_apprch]  ;
3416: WAIT   0.20(sec) ;
3417:L P[2231]  R[157] mm/sec CNT100 TA    0.00sec,CALL RUN_LASER_START Offset,PR[25:Start_Offset] ;
3419:L P[2232]  R[157] mm/sec CNT100 Offset,PR[24:Rotate_Offset] ;
3420:L P[2233]  R[157] mm/sec CNT100 Offset,PR[24:Rotate_Offset] ;
3421:L P[2234]  R[157] mm/sec CNT100 Offset,PR[24:Rotate_Offset] ;
3422:L P[2235]  R[157] mm/sec CNT100 TA    0.00sec,CALL RUN_LASER_STOP Offset,PR[26:Stop_Offset] ;
3424:L P[2235]  R[157] mm/sec FINE Offset,PR[76:Offst_dprt] ;
3425:L P[2236]  R[157] mm/sec CNT100 Offset,PR[24:Rotate_Offset] ;
3426:L P[2237]  R[157] mm/sec CNT100 Offset,PR[24:Rotate_Offset] ;
3427:L P[2238]  R[157] mm/sec CNT100 Offset,PR[24:Rotate_Offset] ;
3428:L P[2239]  R[157] mm/sec CNT100 Offset,PR[24:Rotate_Offset] ;
3429:L P[2240]  R[157] mm/sec CNT100 Offset,PR[24:Rotate_Offset] ;
3430:L P[2241]  R[157] mm/sec CNT100 Offset,PR[24:Rotate_Offset] ;
3431: !Pass169 ;
3432: LBL[1169:Pass169] ;
3433:L P[2242]  R[157] mm/sec FINE Offset,PR[78:Offst_apprch]  ;
3434: WAIT   0.20(sec) ;
3435:L P[2242]  R[157] mm/sec CNT100 TA    0.00sec,CALL RUN_LASER_START Offset,PR[25:Start_Offset] ;
3437:L P[2243]  R[157] mm/sec CNT100 Offset,PR[24:Rotate_Offset] ;
3438:L P[2244]  R[157] mm/sec CNT100 Offset,PR[24:Rotate_Offset] ;
3439:L P[2245]  R[157] mm/sec CNT100 Offset,PR[24:Rotate_Offset] ;
3440:L P[2246]  R[157] mm/sec CNT100 TA    0.00sec,CALL RUN_LASER_STOP Offset,PR[26:Stop_Offset] ;
3442:L P[2246]  R[157] mm/sec FINE Offset,PR[76:Offst_dprt] ;
3443:L P[2247]  R[157] mm/sec CNT100 Offset,PR[24:Rotate_Offset] ;
3444:L P[2248]  R[157] mm/sec CNT100 Offset,PR[24:Rotate_Offset] ;
3445:L P[2249]  R[157] mm/sec CNT100 Offset,PR[24:Rotate_Offset] ;
3446:L P[2250]  R[157] mm/sec CNT100 Offset,PR[24:Rotate_Offset] ;
3447:L P[2251]  R[157] mm/sec CNT100 Offset,PR[24:Rotate_Offset] ;
3448:L P[2252]  R[157] mm/sec CNT100 Offset,PR[24:Rotate_Offset] ;
3449: !Pass170 ;
3450: LBL[1170:Pass170] ;
3451:L P[2253]  R[157] mm/sec FINE Offset,PR[78:Offst_apprch]  ;
3452: WAIT   0.20(sec) ;
3453:L P[2253]  R[157] mm/sec CNT100 TA    0.00sec,CALL RUN_LASER_START Offset,PR[25:Start_Offset] ;
3455:L P[2254]  R[157] mm/sec CNT100 Offset,PR[24:Rotate_Offset] ;
3456:L P[2255]  R[157] mm/sec CNT100 Offset,PR[24:Rotate_Offset] ;
3457:L P[2256]  R[157] mm/sec CNT100 Offset,PR[24:Rotate_Offset] ;
3458:L P[2257]  R[157] mm/sec CNT100 Offset,PR[24:Rotate_Offset] ;
3459:L P[2258]  R[157] mm/sec CNT100 Offset,PR[24:Rotate_Offset] ;
3460:L P[2259]  R[157] mm/sec CNT100 TA    0.00sec,CALL RUN_LASER_STOP Offset,PR[26:Stop_Offset] ;
3462:L P[2259]  R[157] mm/sec FINE Offset,PR[76:Offst_dprt] ;
3463:L P[2260]  R[157] mm/sec CNT100 Offset,PR[24:Rotate_Offset] ;
3464:L P[2261]  R[157] mm/sec CNT100 Offset,PR[24:Rotate_Offset] ;
3465:L P[2262]  R[157] mm/sec CNT100 Offset,PR[24:Rotate_Offset] ;
3466:L P[2263]  R[157] mm/sec CNT100 Offset,PR[24:Rotate_Offset] ;
3467:L P[2264]  R[157] mm/sec CNT100 Offset,PR[24:Rotate_Offset] ;
3468:L P[2265]  R[157] mm/sec CNT100 Offset,PR[24:Rotate_Offset] ;
3469: !Pass171 ;
3470: LBL[1171:Pass171] ;
3471:L P[2266]  R[157] mm/sec FINE Offset,PR[78:Offst_apprch]  ;
3472: WAIT   0.20(sec) ;
3473:L P[2266]  R[157] mm/sec CNT100 TA    0.00sec,CALL RUN_LASER_START Offset,PR[25:Start_Offset] ;
3475:L P[2267]  R[157] mm/sec CNT100 Offset,PR[24:Rotate_Offset] ;
3476:L P[2268]  R[157] mm/sec CNT100 TA    0.00sec,CALL RUN_LASER_STOP Offset,PR[26:Stop_Offset] ;
3478:L P[2268]  R[157] mm/sec FINE Offset,PR[76:Offst_dprt] ;
3479:L P[2269]  R[157] mm/sec CNT100 Offset,PR[24:Rotate_Offset] ;
3480:L P[2270]  R[157] mm/sec CNT100 Offset,PR[24:Rotate_Offset] ;
3481:L P[2271]  R[157] mm/sec CNT100 Offset,PR[24:Rotate_Offset] ;
3482:L P[2272]  R[157] mm/sec CNT100 Offset,PR[24:Rotate_Offset] ;
3483:L P[2273]  R[157] mm/sec CNT100 Offset,PR[24:Rotate_Offset] ;
3484:L P[2274]  R[157] mm/sec CNT100 Offset,PR[24:Rotate_Offset] ;
3485: !Pass172 ;
3486: LBL[1172:Pass172] ;
3487:L P[2275]  R[157] mm/sec FINE Offset,PR[78:Offst_apprch]  ;
3488: WAIT   0.20(sec) ;
3489:L P[2275]  R[157] mm/sec CNT100 TA    0.00sec,CALL RUN_LASER_START Offset,PR[25:Start_Offset] ;
3491:L P[2276]  R[157] mm/sec CNT100 Offset,PR[24:Rotate_Offset] ;
3492:L P[2277]  R[157] mm/sec CNT100 TA    0.00sec,CALL RUN_LASER_STOP Offset,PR[26:Stop_Offset] ;
3494:L P[2277]  R[157] mm/sec FINE Offset,PR[76:Offst_dprt] ;
3495:L P[2278]  R[157] mm/sec CNT100 Offset,PR[24:Rotate_Offset] ;
3496:L P[2279]  R[157] mm/sec CNT100 Offset,PR[24:Rotate_Offset] ;
3497:L P[2280]  R[157] mm/sec CNT100 Offset,PR[24:Rotate_Offset] ;
3498:L P[2281]  R[157] mm/sec CNT100 Offset,PR[24:Rotate_Offset] ;
3499:L P[2282]  R[157] mm/sec CNT100 Offset,PR[24:Rotate_Offset] ;
3500:L P[2283]  R[157] mm/sec CNT100 Offset,PR[24:Rotate_Offset] ;
3501: !Pass173 ;
3502: LBL[1173:Pass173] ;
3503:L P[2284]  R[157] mm/sec FINE Offset,PR[78:Offst_apprch]  ;
3504: WAIT   0.20(sec) ;
3505:L P[2284]  R[157] mm/sec CNT100 TA    0.00sec,CALL RUN_LASER_START Offset,PR[25:Start_Offset] ;
3507:L P[2285]  R[157] mm/sec CNT100 Offset,PR[24:Rotate_Offset] ;
3508:L P[2286]  R[157] mm/sec CNT100 Offset,PR[24:Rotate_Offset] ;
3509:L P[2287]  R[157] mm/sec CNT100 Offset,PR[24:Rotate_Offset] ;
3510:L P[2288]  R[157] mm/sec CNT100 Offset,PR[24:Rotate_Offset] ;
3511:L P[2289]  R[157] mm/sec CNT100 TA    0.00sec,CALL RUN_LASER_STOP Offset,PR[26:Stop_Offset] ;
3513:L P[2289]  R[157] mm/sec FINE Offset,PR[76:Offst_dprt] ;
3514:L P[2290]  R[157] mm/sec CNT100 Offset,PR[24:Rotate_Offset] ;
3515:L P[2291]  R[157] mm/sec CNT100 Offset,PR[24:Rotate_Offset] ;
3516:L P[2292]  R[157] mm/sec CNT100 Offset,PR[24:Rotate_Offset] ;
3517:L P[2293]  R[157] mm/sec CNT100 Offset,PR[24:Rotate_Offset] ;
3518:L P[2294]  R[157] mm/sec CNT100 Offset,PR[24:Rotate_Offset] ;
3519:L P[2295]  R[157] mm/sec CNT100 Offset,PR[24:Rotate_Offset] ;
3520: !Pass174 ;
3521: LBL[1174:Pass174] ;
3522:L P[2296]  R[157] mm/sec FINE Offset,PR[78:Offst_apprch]  ;
3523: WAIT   0.20(sec) ;
3524:L P[2296]  R[157] mm/sec CNT100 TA    0.00sec,CALL RUN_LASER_START Offset,PR[25:Start_Offset] ;
3526:L P[2297]  R[157] mm/sec CNT100 Offset,PR[24:Rotate_Offset] ;
3527:L P[2298]  R[157] mm/sec CNT100 Offset,PR[24:Rotate_Offset] ;
3528:L P[2299]  R[157] mm/sec CNT100 Offset,PR[24:Rotate_Offset] ;
3529:L P[2300]  R[157] mm/sec CNT100 TA    0.00sec,CALL RUN_LASER_STOP Offset,PR[26:Stop_Offset] ;
3531:L P[2300]  R[157] mm/sec FINE Offset,PR[76:Offst_dprt] ;
3532:L P[2301]  R[157] mm/sec CNT100 Offset,PR[24:Rotate_Offset] ;
3533:L P[2302]  R[157] mm/sec CNT100 Offset,PR[24:Rotate_Offset] ;
3534:L P[2303]  R[157] mm/sec CNT100 Offset,PR[24:Rotate_Offset] ;
3535:L P[2304]  R[157] mm/sec CNT100 Offset,PR[24:Rotate_Offset] ;
3536:L P[2305]  R[157] mm/sec CNT100 Offset,PR[24:Rotate_Offset] ;
3537:L P[2306]  R[157] mm/sec CNT100 Offset,PR[24:Rotate_Offset] ;
3538: !Pass175 ;
3539: LBL[1175:Pass175] ;
3540:L P[2307]  R[157] mm/sec FINE Offset,PR[78:Offst_apprch]  ;
3541: WAIT   0.20(sec) ;
3542:L P[2307]  R[157] mm/sec CNT100 TA    0.00sec,CALL RUN_LASER_START Offset,PR[25:Start_Offset] ;
3544:L P[2308]  R[157] mm/sec CNT100 Offset,PR[24:Rotate_Offset] ;
3545:L P[2309]  R[157] mm/sec CNT100 Offset,PR[24:Rotate_Offset] ;
3546:L P[2310]  R[157] mm/sec CNT100 Offset,PR[24:Rotate_Offset] ;
3547:L P[2311]  R[157] mm/sec CNT100 TA    0.00sec,CALL RUN_LASER_STOP Offset,PR[26:Stop_Offset] ;
3549:L P[2311]  R[157] mm/sec FINE Offset,PR[76:Offst_dprt] ;
3550:L P[2312]  R[157] mm/sec CNT100 Offset,PR[24:Rotate_Offset] ;
3551:L P[2313]  R[157] mm/sec CNT100 Offset,PR[24:Rotate_Offset] ;
